REGION Network 16: Odczyt 30011
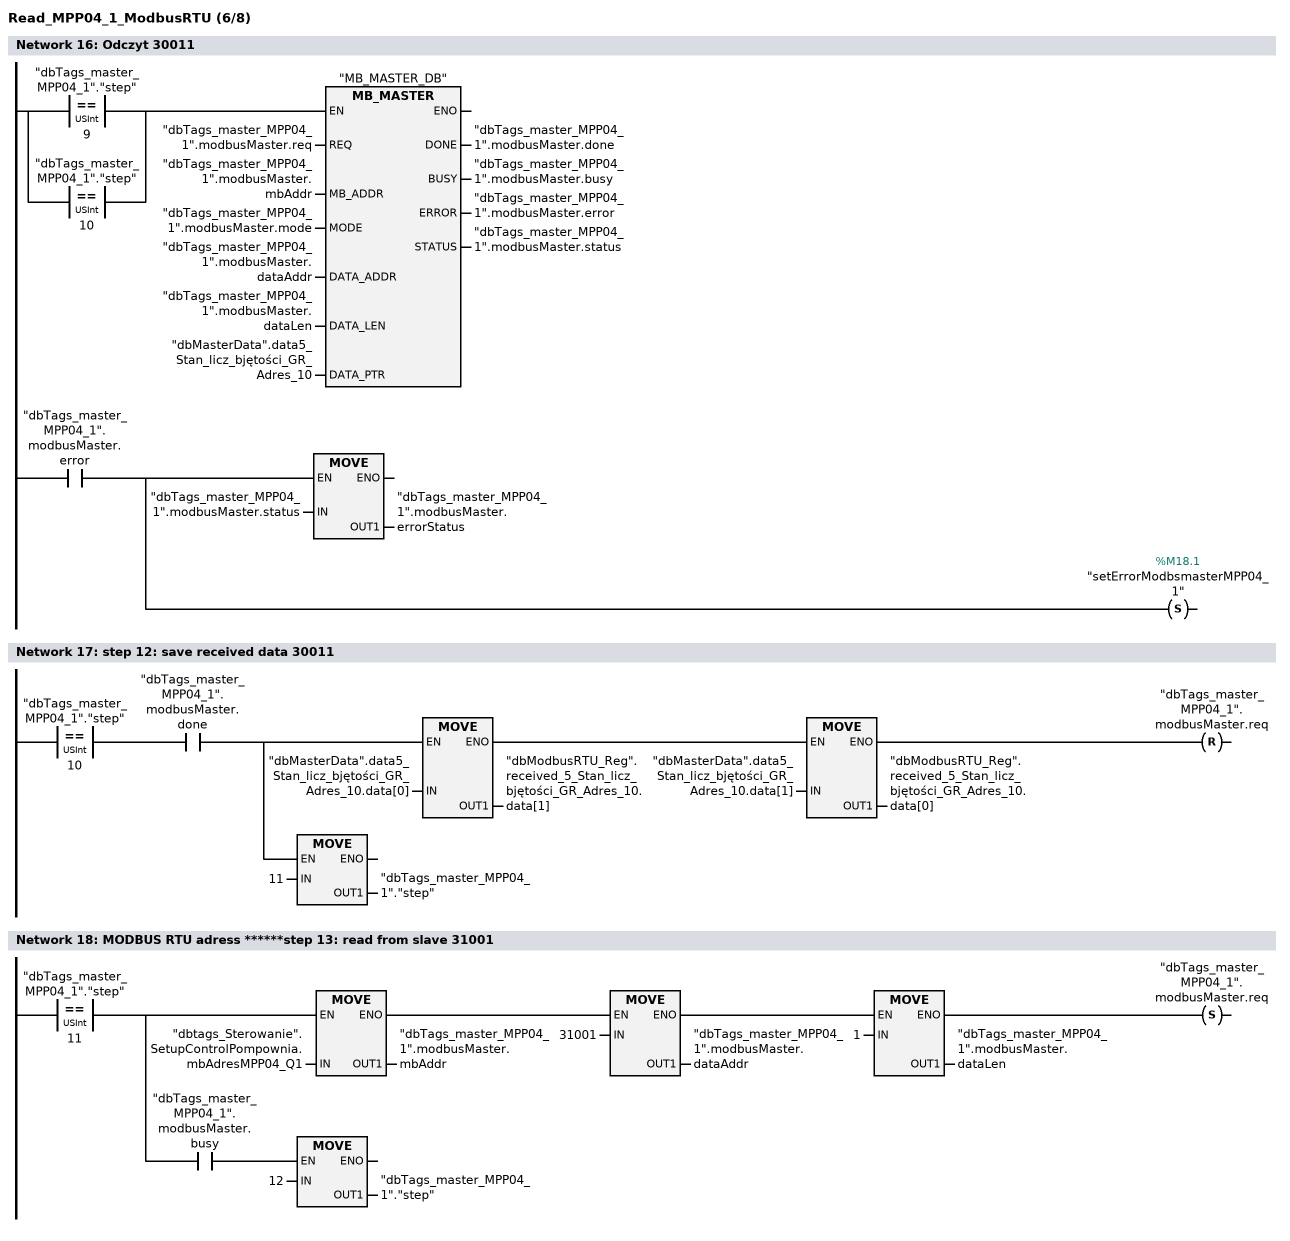
   RUNG wire#powerrail
      { S7_Templates := "SrcType := USInt" } EQ_Contact(in1 := "dbTags_master_MPP04_1"."step", in2 := 9)
      wire#w1
      "MB_MASTER_DB".MB_MASTER(REQ := "dbTags_master_MPP04_1".modbusMaster.req, MB_ADDR := "dbTags_master_MPP04_1".modbusMaster.mbAddr, MODE := "dbTags_master_MPP04_1".modbusMaster.mode, DATA_ADDR := "dbTags_master_MPP04_1".modbusMaster.dataAddr, DATA_LEN := "dbTags_master_MPP04_1".modbusMaster.dataLen, DATA_PTR := "dbMasterData".data5_Stan_licz_bjętości_GR_Adres_10, DONE => "dbTags_master_MPP04_1".modbusMaster.done, BUSY => "dbTags_master_MPP04_1".modbusMaster.busy, ERROR => "dbTags_master_MPP04_1".modbusMaster.error, STATUS => "dbTags_master_MPP04_1".modbusMaster.status)
   END_RUNG
   RUNG wire#powerrail
      { S7_Templates := "SrcType := USInt" } EQ_Contact(in1 := "dbTags_master_MPP04_1"."step", in2 := 10)
   END_RUNG wire#w1
   RUNG wire#powerrail
      Contact( "dbTags_master_MPP04_1".modbusMaster.error )
      wire#w2
      { S7_GenerateENO := "TRUE" } Move(in := "dbTags_master_MPP04_1".modbusMaster.status, out1 => "dbTags_master_MPP04_1".modbusMaster.errorStatus)
   END_RUNG
   RUNG wire#w2
      S_Coil( "setErrorModbsmasterMPP04_1" )
   END_RUNG
   // the same network as SCL:
   IF ("dbTags_master_MPP04_1"."step" = 9) OR ("dbTags_master_MPP04_1"."step" = 10) THEN
       "MB_MASTER_DB"(REQ := "dbTags_master_MPP04_1".modbusMaster.req,   // MB_MASTER
                      MB_ADDR := "dbTags_master_MPP04_1".modbusMaster.mbAddr,
                      MODE := "dbTags_master_MPP04_1".modbusMaster.mode,
                      DATA_ADDR := "dbTags_master_MPP04_1".modbusMaster.dataAddr,
                      DATA_LEN := "dbTags_master_MPP04_1".modbusMaster.dataLen,
                      DATA_PTR := "dbMasterData".data5_Stan_licz_bjętości_GR_Adres_10,
                      DONE => "dbTags_master_MPP04_1".modbusMaster.done,
                      BUSY => "dbTags_master_MPP04_1".modbusMaster.busy,
                      ERROR => "dbTags_master_MPP04_1".modbusMaster.error,
                      STATUS => "dbTags_master_MPP04_1".modbusMaster.status);
   END_IF;
   IF "dbTags_master_MPP04_1".modbusMaster.error THEN
       "dbTags_master_MPP04_1".modbusMaster.errorStatus := "dbTags_master_MPP04_1".modbusMaster.status;
       "setErrorModbsmasterMPP04_1" := TRUE;
   END_IF;
END_REGION

REGION Network 17: step 12: save received data 30011
   RUNG wire#powerrail
      { S7_Templates := "SrcType := USInt" } EQ_Contact(in1 := "dbTags_master_MPP04_1"."step", in2 := 10)
      Contact( "dbTags_master_MPP04_1".modbusMaster.done )
      wire#w1
      { S7_GenerateENO := "TRUE" } Move(in := "dbMasterData".data5_Stan_licz_bjętości_GR_Adres_10.data[0], out1 => "dbModbusRTU_Reg".received_5_Stan_licz_bjętości_GR_Adres_10.data[1])
      { S7_GenerateENO := "TRUE" } Move(in := "dbMasterData".data5_Stan_licz_bjętości_GR_Adres_10.data[1], out1 => "dbModbusRTU_Reg".received_5_Stan_licz_bjętości_GR_Adres_10.data[0])
      R_Coil( "dbTags_master_MPP04_1".modbusMaster.req )
   END_RUNG
   RUNG wire#w1
      { S7_GenerateENO := "TRUE" } Move(in := 11, out1 => "dbTags_master_MPP04_1"."step")
   END_RUNG
   // the same network as SCL:
   // ENO of a box is taken as its EN; it also drops when the box reports an error
   IF ("dbTags_master_MPP04_1"."step" = 10) AND "dbTags_master_MPP04_1".modbusMaster.done THEN
       "dbModbusRTU_Reg".received_5_Stan_licz_bjętości_GR_Adres_10.data[1] := "dbMasterData".data5_Stan_licz_bjętości_GR_Adres_10.data[0];
       "dbModbusRTU_Reg".received_5_Stan_licz_bjętości_GR_Adres_10.data[0] := "dbMasterData".data5_Stan_licz_bjętości_GR_Adres_10.data[1];
       "dbTags_master_MPP04_1".modbusMaster.req := FALSE;
       "dbTags_master_MPP04_1"."step" := 11;
   END_IF;
END_REGION

REGION Network 18: MODBUS RTU adress ******step 13: read from slave 31001
   RUNG wire#powerrail
      { S7_Templates := "SrcType := USInt" } EQ_Contact(in1 := "dbTags_master_MPP04_1"."step", in2 := 11)
      wire#w1
      Move(in := "dbtags_Sterowanie".SetupControlPompownia.mbAdresMPP04_Q1, out1 => "dbTags_master_MPP04_1".modbusMaster.mbAddr)
      { S7_GenerateENO := "TRUE" } Move(in := 31001, out1 => "dbTags_master_MPP04_1".modbusMaster.dataAddr)
      Move(in := 1, out1 => "dbTags_master_MPP04_1".modbusMaster.dataLen)
      S_Coil( "dbTags_master_MPP04_1".modbusMaster.req )
   END_RUNG
   RUNG wire#w1
      Contact( "dbTags_master_MPP04_1".modbusMaster.busy )
      { S7_GenerateENO := "TRUE" } Move(in := 12, out1 => "dbTags_master_MPP04_1"."step")
   END_RUNG
   // the same network as SCL:
   // ENO of a box is taken as its EN; it also drops when the box reports an error
   #_w1 := "dbTags_master_MPP04_1"."step" = 11;
   IF #_w1 THEN
       "dbTags_master_MPP04_1".modbusMaster.mbAddr := "dbtags_Sterowanie".SetupControlPompownia.mbAdresMPP04_Q1;
       "dbTags_master_MPP04_1".modbusMaster.dataAddr := 31001;
       "dbTags_master_MPP04_1".modbusMaster.dataLen := 1;
       "dbTags_master_MPP04_1".modbusMaster.req := TRUE;
   END_IF;
   IF #_w1 AND "dbTags_master_MPP04_1".modbusMaster.busy THEN "dbTags_master_MPP04_1"."step" := 12; END_IF;
END_REGION

REGION Network 19: Odcztyt 31001
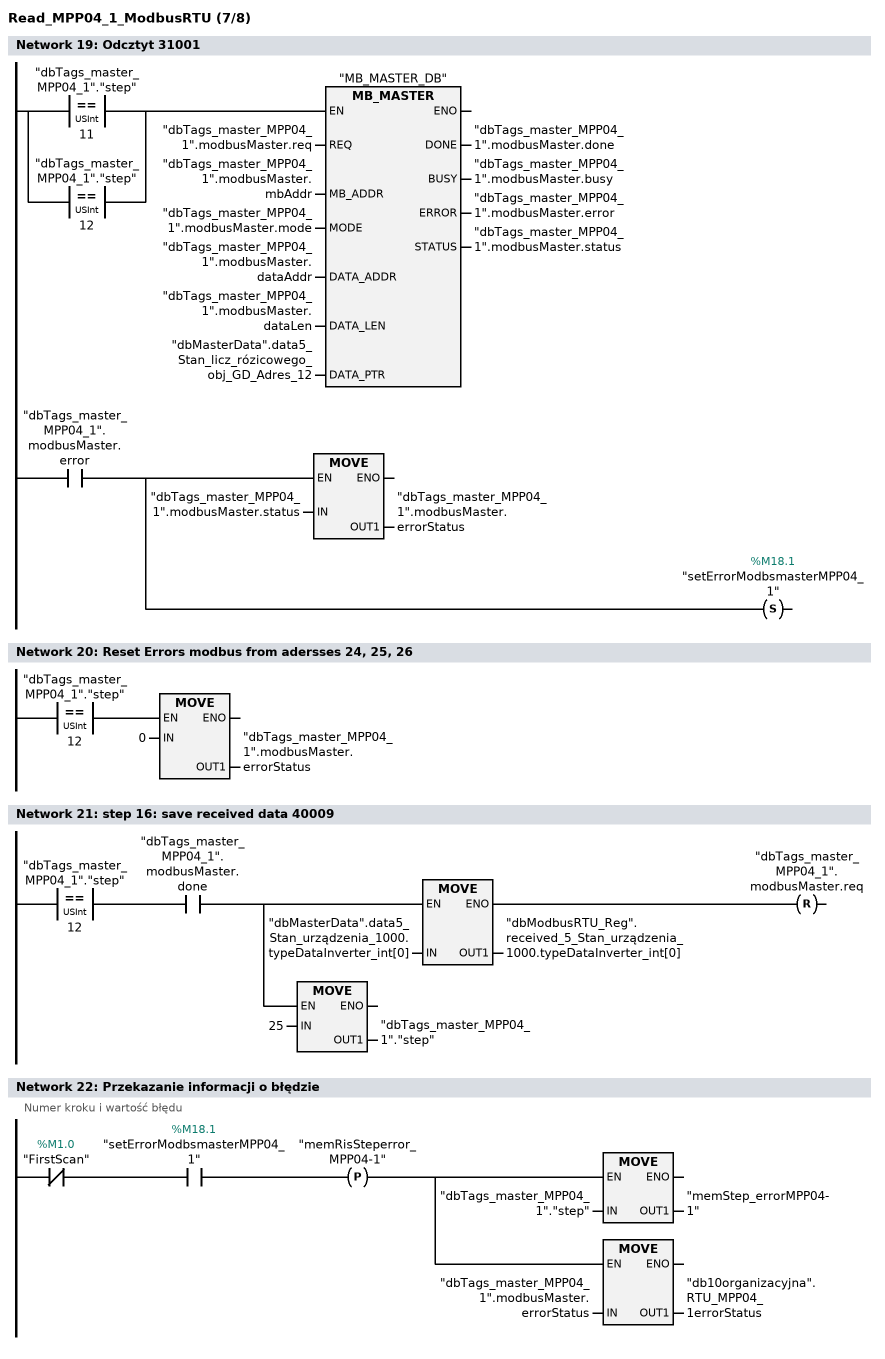
   RUNG wire#powerrail
      { S7_Templates := "SrcType := USInt" } EQ_Contact(in1 := "dbTags_master_MPP04_1"."step", in2 := 11)
      wire#w1
      "MB_MASTER_DB".MB_MASTER(REQ := "dbTags_master_MPP04_1".modbusMaster.req, MB_ADDR := "dbTags_master_MPP04_1".modbusMaster.mbAddr, MODE := "dbTags_master_MPP04_1".modbusMaster.mode, DATA_ADDR := "dbTags_master_MPP04_1".modbusMaster.dataAddr, DATA_LEN := "dbTags_master_MPP04_1".modbusMaster.dataLen, DATA_PTR := "dbMasterData".data5_Stan_licz_rózicowego_obj_GD_Adres_12, DONE => "dbTags_master_MPP04_1".modbusMaster.done, BUSY => "dbTags_master_MPP04_1".modbusMaster.busy, ERROR => "dbTags_master_MPP04_1".modbusMaster.error, STATUS => "dbTags_master_MPP04_1".modbusMaster.status)
   END_RUNG
   RUNG wire#powerrail
      { S7_Templates := "SrcType := USInt" } EQ_Contact(in1 := "dbTags_master_MPP04_1"."step", in2 := 12)
   END_RUNG wire#w1
   RUNG wire#powerrail
      Contact( "dbTags_master_MPP04_1".modbusMaster.error )
      wire#w2
      { S7_GenerateENO := "TRUE" } Move(in := "dbTags_master_MPP04_1".modbusMaster.status, out1 => "dbTags_master_MPP04_1".modbusMaster.errorStatus)
   END_RUNG
   RUNG wire#w2
      S_Coil( "setErrorModbsmasterMPP04_1" )
   END_RUNG
   // the same network as SCL:
   IF ("dbTags_master_MPP04_1"."step" = 11) OR ("dbTags_master_MPP04_1"."step" = 12) THEN
       "MB_MASTER_DB"(REQ := "dbTags_master_MPP04_1".modbusMaster.req,   // MB_MASTER
                      MB_ADDR := "dbTags_master_MPP04_1".modbusMaster.mbAddr,
                      MODE := "dbTags_master_MPP04_1".modbusMaster.mode,
                      DATA_ADDR := "dbTags_master_MPP04_1".modbusMaster.dataAddr,
                      DATA_LEN := "dbTags_master_MPP04_1".modbusMaster.dataLen,
                      DATA_PTR := "dbMasterData".data5_Stan_licz_rózicowego_obj_GD_Adres_12,
                      DONE => "dbTags_master_MPP04_1".modbusMaster.done,
                      BUSY => "dbTags_master_MPP04_1".modbusMaster.busy,
                      ERROR => "dbTags_master_MPP04_1".modbusMaster.error,
                      STATUS => "dbTags_master_MPP04_1".modbusMaster.status);
   END_IF;
   IF "dbTags_master_MPP04_1".modbusMaster.error THEN
       "dbTags_master_MPP04_1".modbusMaster.errorStatus := "dbTags_master_MPP04_1".modbusMaster.status;
       "setErrorModbsmasterMPP04_1" := TRUE;
   END_IF;
END_REGION

REGION Network 20: Reset Errors modbus from adersses 24, 25, 26
   RUNG wire#powerrail
      { S7_Templates := "SrcType := USInt" } EQ_Contact(in1 := "dbTags_master_MPP04_1"."step", in2 := 12)
      { S7_GenerateENO := "TRUE" } Move(in := 0, out1 => "dbTags_master_MPP04_1".modbusMaster.errorStatus)
   END_RUNG
   // the same network as SCL:
   IF "dbTags_master_MPP04_1"."step" = 12 THEN "dbTags_master_MPP04_1".modbusMaster.errorStatus := 0; END_IF;
END_REGION

REGION Network 21: step 16: save received data 40009
   RUNG wire#powerrail
      { S7_Templates := "SrcType := USInt" } EQ_Contact(in1 := "dbTags_master_MPP04_1"."step", in2 := 12)
      Contact( "dbTags_master_MPP04_1".modbusMaster.done )
      wire#w1
      { S7_GenerateENO := "TRUE" } Move(in := "dbMasterData".data5_Stan_urządzenia_1000.typeDataInverter_int[0], out1 => "dbModbusRTU_Reg".received_5_Stan_urządzenia_1000.typeDataInverter_int[0])
      R_Coil( "dbTags_master_MPP04_1".modbusMaster.req )
   END_RUNG
   RUNG wire#w1
      { S7_GenerateENO := "TRUE" } Move(in := 25, out1 => "dbTags_master_MPP04_1"."step")
   END_RUNG
   // the same network as SCL:
   // ENO of a box is taken as its EN; it also drops when the box reports an error
   IF ("dbTags_master_MPP04_1"."step" = 12) AND "dbTags_master_MPP04_1".modbusMaster.done THEN
       "dbModbusRTU_Reg".received_5_Stan_urządzenia_1000.typeDataInverter_int[0] := "dbMasterData".data5_Stan_urządzenia_1000.typeDataInverter_int[0];
       "dbTags_master_MPP04_1".modbusMaster.req := FALSE;
       "dbTags_master_MPP04_1"."step" := 25;
   END_IF;
END_REGION

REGION Network 22: Przekazanie informacji o błędzie
   // Numer kroku i wartość błędu
   RUNG wire#powerrail
      I_Contact( "FirstScan" )
      Contact( "setErrorModbsmasterMPP04_1" )
      P_Trig( "memRisSteperror_MPP04-1" )
      wire#w1
      Move(in := "dbTags_master_MPP04_1"."step", out1 => "memStep_errorMPP04-1")
   END_RUNG
   RUNG wire#w1
      { S7_GenerateENO := "TRUE" } Move(in := "dbTags_master_MPP04_1".modbusMaster.errorStatus, out1 => "db10organizacyjna".RTU_MPP04_1errorStatus)
   END_RUNG
   // the same network as SCL:
   #_w1 := NOT "FirstScan" AND "setErrorModbsmasterMPP04_1";
   #_w2 := #_w1 AND NOT "memRisSteperror_MPP04-1";   // rising edge
   "memRisSteperror_MPP04-1" := #_w1;
   IF #_w2 THEN
       "memStep_errorMPP04-1" := "dbTags_master_MPP04_1"."step";
       "db10organizacyjna".RTU_MPP04_1errorStatus := "dbTags_master_MPP04_1".modbusMaster.errorStatus;
   END_IF;
END_REGION

REGION Network 23: Obsługa błędów Modbaus
   // Inicjacja pętli modbus dla następnego urządzenia
   // Ustawienie kroku pętli na stan awaria [27]
   // Uwolnienie linni modbus
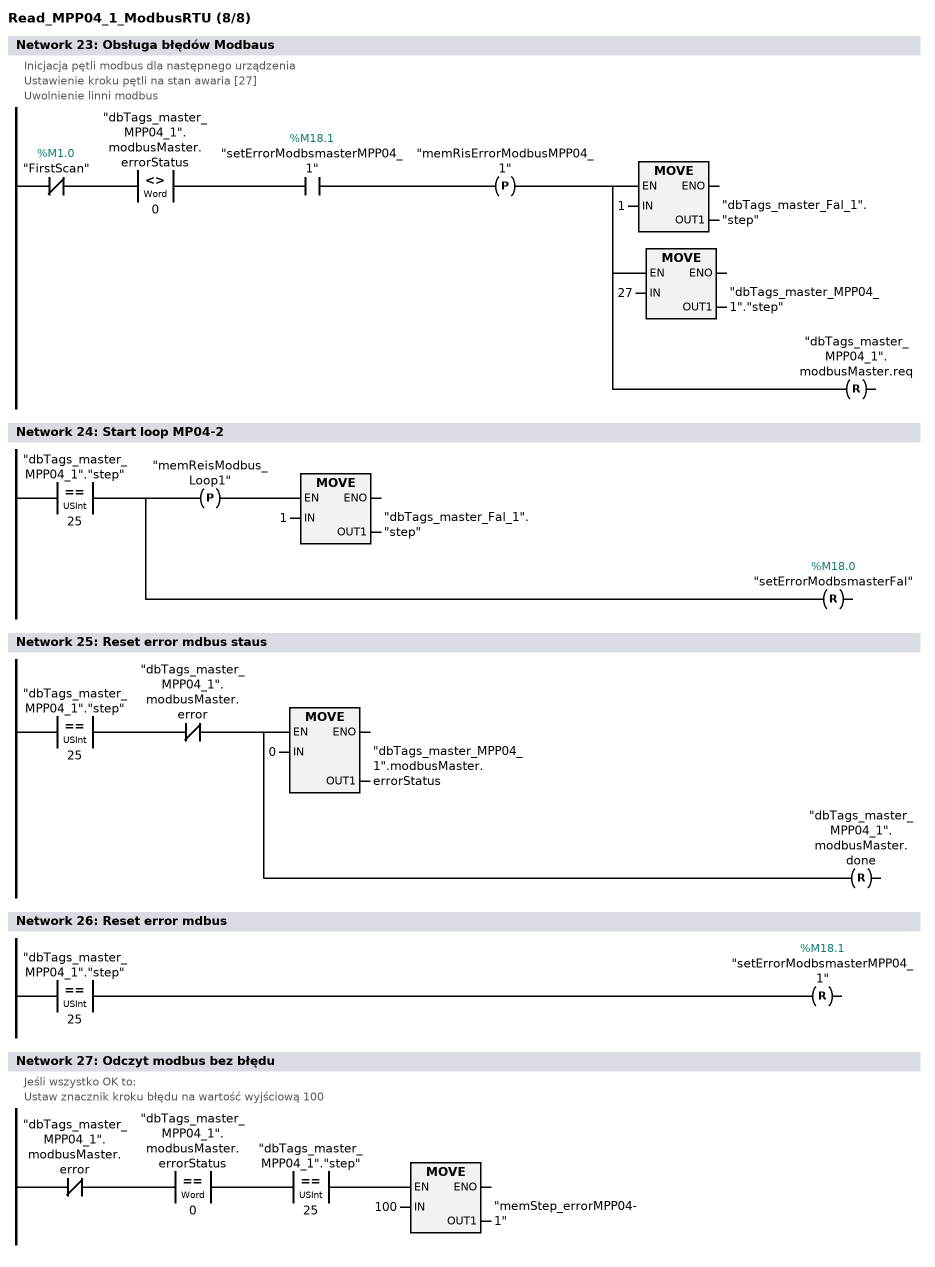
   RUNG wire#powerrail
      I_Contact( "FirstScan" )
      { S7_Templates := "SrcType := Word" } NE_Contact(in1 := "dbTags_master_MPP04_1".modbusMaster.errorStatus, in2 := 0)
      Contact( "setErrorModbsmasterMPP04_1" )
      P_Trig( "memRisErrorModbusMPP04_1" )
      wire#w1
      { S7_GenerateENO := "TRUE" } Move(in := 1, out1 => "dbTags_master_Fal_1"."step")
   END_RUNG
   RUNG wire#w1
      { S7_GenerateENO := "TRUE" } Move(in := 27, out1 => "dbTags_master_MPP04_1"."step")
   END_RUNG
   RUNG wire#w1
      R_Coil( "dbTags_master_MPP04_1".modbusMaster.req )
   END_RUNG
   // the same network as SCL:
   #_w1 := NOT "FirstScan" AND ("dbTags_master_MPP04_1".modbusMaster.errorStatus <> 0) AND "setErrorModbsmasterMPP04_1";
   #_w2 := #_w1 AND NOT "memRisErrorModbusMPP04_1";   // rising edge
   "memRisErrorModbusMPP04_1" := #_w1;
   IF #_w2 THEN
       "dbTags_master_Fal_1"."step" := 1;
       "dbTags_master_MPP04_1"."step" := 27;
       "dbTags_master_MPP04_1".modbusMaster.req := FALSE;
   END_IF;
END_REGION

REGION Network 24: Start loop MP04-2
   RUNG wire#powerrail
      { S7_Templates := "SrcType := USInt" } EQ_Contact(in1 := "dbTags_master_MPP04_1"."step", in2 := 25)
      wire#w1
      P_Trig( "memReisModbus_Loop1" )
      { S7_GenerateENO := "TRUE" } Move(in := 1, out1 => "dbTags_master_Fal_1"."step")
   END_RUNG
   RUNG wire#w1
      R_Coil( "setErrorModbsmasterFal" )
   END_RUNG
   // the same network as SCL:
   #_w1 := "dbTags_master_MPP04_1"."step" = 25;
   #_w2 := #_w1 AND NOT "memReisModbus_Loop1";   // rising edge
   "memReisModbus_Loop1" := #_w1;
   IF #_w2 THEN "dbTags_master_Fal_1"."step" := 1; END_IF;
   IF #_w1 THEN "setErrorModbsmasterFal" := FALSE; END_IF;
END_REGION

REGION Network 25: Reset error mdbus staus
   RUNG wire#powerrail
      { S7_Templates := "SrcType := USInt" } EQ_Contact(in1 := "dbTags_master_MPP04_1"."step", in2 := 25)
      I_Contact( "dbTags_master_MPP04_1".modbusMaster.error )
      wire#w1
      { S7_GenerateENO := "TRUE" } Move(in := 0, out1 => "dbTags_master_MPP04_1".modbusMaster.errorStatus)
   END_RUNG
   RUNG wire#w1
      R_Coil( "dbTags_master_MPP04_1".modbusMaster.done )
   END_RUNG
   // the same network as SCL:
   IF ("dbTags_master_MPP04_1"."step" = 25) AND NOT "dbTags_master_MPP04_1".modbusMaster.error THEN
       "dbTags_master_MPP04_1".modbusMaster.errorStatus := 0;
       "dbTags_master_MPP04_1".modbusMaster.done := FALSE;
   END_IF;
END_REGION

REGION Network 26: Reset error mdbus
   RUNG wire#powerrail
      { S7_Templates := "SrcType := USInt" } EQ_Contact(in1 := "dbTags_master_MPP04_1"."step", in2 := 25)
      R_Coil( "setErrorModbsmasterMPP04_1" )
   END_RUNG
   // the same network as SCL:
   IF "dbTags_master_MPP04_1"."step" = 25 THEN "setErrorModbsmasterMPP04_1" := FALSE; END_IF;
END_REGION

REGION Network 27: Odczyt modbus bez błędu
   // Jeśli wszystko OK to:
   // Ustaw znacznik kroku błędu na wartość wyjściową 100
   RUNG wire#powerrail
      I_Contact( "dbTags_master_MPP04_1".modbusMaster.error )
      { S7_Templates := "SrcType := Word" } EQ_Contact(in1 := "dbTags_master_MPP04_1".modbusMaster.errorStatus, in2 := 0)
      { S7_Templates := "SrcType := USInt" } EQ_Contact(in1 := "dbTags_master_MPP04_1"."step", in2 := 25)
      { S7_GenerateENO := "TRUE" } Move(in := 100, out1 => "memStep_errorMPP04-1")
   END_RUNG
   // the same network as SCL:
   IF NOT "dbTags_master_MPP04_1".modbusMaster.error AND ("dbTags_master_MPP04_1".modbusMaster.errorStatus = 0) AND ("dbTags_master_MPP04_1"."step" = 25) THEN
       "memStep_errorMPP04-1" := 100;
   END_IF;
END_REGION
END_FUNCTION

FUNCTION_BLOCK "Write_dbHold_TCP_Sending"
{ S7_Optimized_Access := 'TRUE' }
VERSION : 0.1

BEGIN
	(*
	
	*)
	
	
	
	
	REGION Strategia Sterowania Pompownią 
	  // przekazanie wartości do PLC2 Zbiorniki
	  "dbHold_RRG".Sending.set_strategia_sterowania:= "dbHoldRegSlave_to_MT101".instSygSter_1;
	  
	END_REGION
	
	REGION _name_
	  // 
	
	
	  
	  
	END_REGION
	
	
	
END_FUNCTION_BLOCK

FUNCTION "Blok liczników pracy" : Void   // FC8, LAD
TITLE = Wywołanie funkcji liczników pracy
{ S7_Optimized_Access := 'TRUE' }
AUTHOR : RTecmer
VERSION : 0.1
// Funkcja wywołuje liczniki pracy napędów
// stored: AutoNumber true, IsIECCheckEnabled false, SetENOAutomatically false, UDAEnableTagReadback false
BEGIN

REGION Network 1: Pompa P1
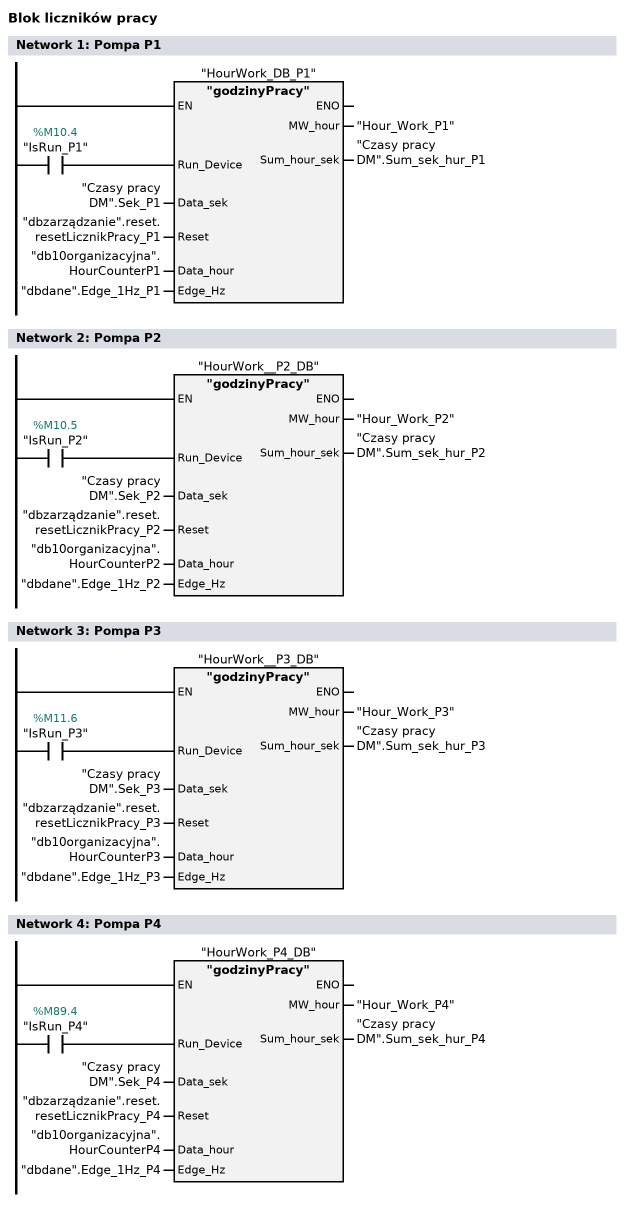
   RUNG wire#powerrail
      "HourWork_DB_P1"(Run_Device := wire#w1, Data_sek := "Czasy pracy DM".Sek_P1, Reset := "dbzarządzanie".reset.resetLicznikPracy_P1, Data_hour := "db10organizacyjna".HourCounterP1, Edge_Hz := "dbdane".Edge_1Hz_P1, MW_hour => "Hour_Work_P1", Sum_hour_sek => "Czasy pracy DM".Sum_sek_hur_P1)
   END_RUNG
   RUNG wire#powerrail
      Contact( "IsRun_P1" )
   END_RUNG wire#w1
   // the same network as SCL:
   "HourWork_DB_P1"(Run_Device := "IsRun_P1",   // "godzinyPracy"
                    Data_sek := "Czasy pracy DM".Sek_P1,
                    Reset := "dbzarządzanie".reset.resetLicznikPracy_P1,
                    Data_hour := "db10organizacyjna".HourCounterP1,
                    Edge_Hz := "dbdane".Edge_1Hz_P1,
                    MW_hour => "Hour_Work_P1",
                    Sum_hour_sek => "Czasy pracy DM".Sum_sek_hur_P1);
END_REGION

REGION Network 2: Pompa P2
   RUNG wire#powerrail
      "HourWork__P2_DB"(Run_Device := wire#w1, Data_sek := "Czasy pracy DM".Sek_P2, Reset := "dbzarządzanie".reset.resetLicznikPracy_P2, Data_hour := "db10organizacyjna".HourCounterP2, Edge_Hz := "dbdane".Edge_1Hz_P2, MW_hour => "Hour_Work_P2", Sum_hour_sek => "Czasy pracy DM".Sum_sek_hur_P2)
   END_RUNG
   RUNG wire#powerrail
      Contact( "IsRun_P2" )
   END_RUNG wire#w1
   // the same network as SCL:
   "HourWork__P2_DB"(Run_Device := "IsRun_P2",   // "godzinyPracy"
                     Data_sek := "Czasy pracy DM".Sek_P2,
                     Reset := "dbzarządzanie".reset.resetLicznikPracy_P2,
                     Data_hour := "db10organizacyjna".HourCounterP2,
                     Edge_Hz := "dbdane".Edge_1Hz_P2,
                     MW_hour => "Hour_Work_P2",
                     Sum_hour_sek => "Czasy pracy DM".Sum_sek_hur_P2);
END_REGION

REGION Network 3: Pompa P3
   RUNG wire#powerrail
      "HourWork__P3_DB"(Run_Device := wire#w1, Data_sek := "Czasy pracy DM".Sek_P3, Reset := "dbzarządzanie".reset.resetLicznikPracy_P3, Data_hour := "db10organizacyjna".HourCounterP3, Edge_Hz := "dbdane".Edge_1Hz_P3, MW_hour => "Hour_Work_P3", Sum_hour_sek => "Czasy pracy DM".Sum_sek_hur_P3)
   END_RUNG
   RUNG wire#powerrail
      Contact( "IsRun_P3" )
   END_RUNG wire#w1
   // the same network as SCL:
   "HourWork__P3_DB"(Run_Device := "IsRun_P3",   // "godzinyPracy"
                     Data_sek := "Czasy pracy DM".Sek_P3,
                     Reset := "dbzarządzanie".reset.resetLicznikPracy_P3,
                     Data_hour := "db10organizacyjna".HourCounterP3,
                     Edge_Hz := "dbdane".Edge_1Hz_P3,
                     MW_hour => "Hour_Work_P3",
                     Sum_hour_sek => "Czasy pracy DM".Sum_sek_hur_P3);
END_REGION

REGION Network 4: Pompa P4
   RUNG wire#powerrail
      "HourWork_P4_DB"(Run_Device := wire#w1, Data_sek := "Czasy pracy DM".Sek_P4, Reset := "dbzarządzanie".reset.resetLicznikPracy_P4, Data_hour := "db10organizacyjna".HourCounterP4, Edge_Hz := "dbdane".Edge_1Hz_P4, MW_hour => "Hour_Work_P4", Sum_hour_sek => "Czasy pracy DM".Sum_sek_hur_P4)
   END_RUNG
   RUNG wire#powerrail
      Contact( "IsRun_P4" )
   END_RUNG wire#w1
   // the same network as SCL:
   "HourWork_P4_DB"(Run_Device := "IsRun_P4",   // "godzinyPracy"
                    Data_sek := "Czasy pracy DM".Sek_P4,
                    Reset := "dbzarządzanie".reset.resetLicznikPracy_P4,
                    Data_hour := "db10organizacyjna".HourCounterP4,
                    Edge_Hz := "dbdane".Edge_1Hz_P4,
                    MW_hour => "Hour_Work_P4",
                    Sum_hour_sek => "Czasy pracy DM".Sum_sek_hur_P4);
END_REGION
END_FUNCTION

FUNCTION_BLOCK "godzinyPracy"   // FB2, LAD
{ S7_Optimized_Access := 'TRUE' }
AUTHOR : RTecmer
FAMILY : XMHour
VERSION : 0.1
// Licznik czasu pracy
// stored: AutoNumber true, IsIECCheckEnabled false, IsRetainMemResEnabled false, MemoryReserve 500, SetENOAutomatically false, UDAEnableTagReadback false
   VAR_INPUT
      Run_Device : Bool;
   END_VAR
   VAR_OUTPUT
      MW_hour : DWord;
      Sum_hour_sek : Real;   // Licznik sumator godzin i sekund na potrzeby wyznaczania dumchawy do pracy
   END_VAR
   VAR_IN_OUT
      Data_sek : Int;
      Reset { ExternalAccessible := 'False'; ExternalVisible := 'False'; ExternalWritable := 'False'} : Bool;
      Data_hour : DWord;
      Edge_Hz { ExternalAccessible := 'False'; ExternalVisible := 'False'; ExternalWritable := 'False'} : Bool;
   END_VAR
   VAR
      sek_real { ExternalAccessible := 'False'; ExternalVisible := 'False'; ExternalWritable := 'False'} : Real;   // pomocnicza konwerski sekund
      actSekReal { ExternalAccessible := 'False'; ExternalVisible := 'False'; ExternalWritable := 'False'} : Real;   // aktualne sekundy po konwersji
      hour_sek { ExternalAccessible := 'False'; ExternalVisible := 'False'; ExternalWritable := 'False'} : Real;
   END_VAR
   VAR_TEMP   // added for the SCL form of the ladder/FBD networks
      _w1 : Bool;
      _w2 : Bool;
   END_VAR
BEGIN

REGION Network 1
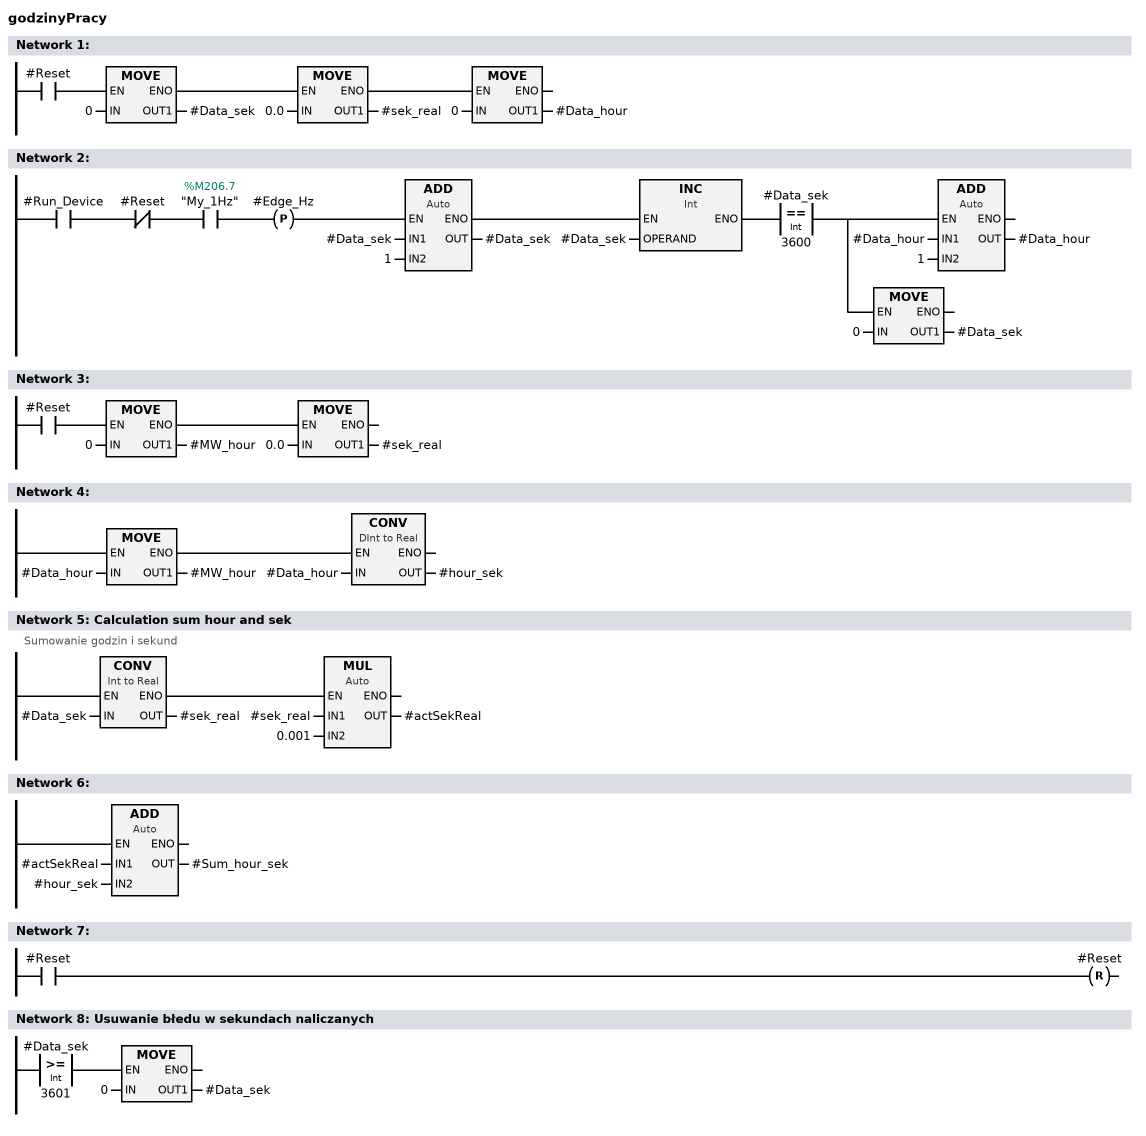
   RUNG wire#powerrail
      Contact( #Reset )
      { S7_GenerateENO := "TRUE" } Move(in := 0, out1 => #Data_sek)
      { S7_GenerateENO := "TRUE" } Move(in := 0.0, out1 => #sek_real)
      { S7_GenerateENO := "TRUE" } Move(in := 0, out1 => #Data_hour)
   END_RUNG
   // the same network as SCL:
   // ENO of a box is taken as its EN; it also drops when the box reports an error
   IF #Reset THEN
       #Data_sek := 0;
       #sek_real := 0.0;
       #Data_hour := 0;
   END_IF;
END_REGION

REGION Network 2
   RUNG wire#powerrail
      Contact( #Run_Device )
      I_Contact( #Reset )
      Contact( "My_1Hz" )
      P_Trig( #Edge_Hz )
      { S7_GenerateENO := "TRUE" } Add(in1 := #Data_sek, in2 := 1, out => #Data_sek)
      { S7_Templates := "DestType := Int"; S7_GenerateENO := "TRUE" } Inc( #Data_sek )
      { S7_Templates := "SrcType := Int" } EQ_Contact(in1 := #Data_sek, in2 := 3600)
      wire#w1
      { S7_GenerateENO := "TRUE" } Add(in1 := #Data_hour, in2 := 1, out => #Data_hour)
   END_RUNG
   RUNG wire#w1
      { S7_GenerateENO := "TRUE" } Move(in := 0, out1 => #Data_sek)
   END_RUNG
   // the same network as SCL:
   // ENO of a box is taken as its EN; it also drops when the box reports an error
   #_w1 := #Run_Device AND NOT #Reset AND "My_1Hz";
   #_w2 := #_w1 AND NOT #Edge_Hz;   // rising edge
   #Edge_Hz := #_w1;
   IF #_w2 THEN
       #Data_sek := #Data_sek + 1;
       #Data_sek := #Data_sek + 1;
   END_IF;
   IF #_w2 AND (#Data_sek = 3600) THEN
       #Data_hour := #Data_hour + 1;
       #Data_sek := 0;
   END_IF;
END_REGION

REGION Network 3
   RUNG wire#powerrail
      Contact( #Reset )
      { S7_GenerateENO := "TRUE" } Move(in := 0, out1 => #MW_hour)
      { S7_GenerateENO := "TRUE" } Move(in := 0.0, out1 => #sek_real)
   END_RUNG
   // the same network as SCL:
   // ENO of a box is taken as its EN; it also drops when the box reports an error
   IF #Reset THEN
       #MW_hour := 0;
       #sek_real := 0.0;
   END_IF;
END_REGION

REGION Network 4
   RUNG wire#powerrail
      { S7_GenerateENO := "TRUE" } Move(in := #Data_hour, out1 => #MW_hour)
      { S7_Templates := "[SrcType := DInt, DestType := Real]" } Convert(in := #Data_hour, out => #hour_sek)
   END_RUNG
   // the same network as SCL:
   // ENO of a box is taken as its EN; it also drops when the box reports an error
   #MW_hour := #Data_hour;
   #hour_sek := DINT_TO_REAL(#Data_hour);
END_REGION

REGION Network 5: Calculation sum hour and sek
   // Sumowanie godzin i sekund
   RUNG wire#powerrail
      { S7_Templates := "[SrcType := Int, DestType := Real]" } Convert(in := #Data_sek, out => #sek_real)
      Mul(in1 := #sek_real, in2 := 0.001, out => #actSekReal)
   END_RUNG
   // the same network as SCL:
   #sek_real := INT_TO_REAL(#Data_sek);
   #actSekReal := #sek_real * 0.001;
END_REGION

REGION Network 6
   RUNG wire#powerrail
      Add(in1 := #actSekReal, in2 := #hour_sek, out => #Sum_hour_sek)
   END_RUNG
   // the same network as SCL:
   #Sum_hour_sek := #actSekReal + #hour_sek;
END_REGION

REGION Network 7
   RUNG wire#powerrail
      Contact( #Reset )
      R_Coil( #Reset )
   END_RUNG
   // the same network as SCL:
   IF #Reset THEN #Reset := FALSE; END_IF;
END_REGION

REGION Network 8: Usuwanie błedu w sekundach naliczanych
   RUNG wire#powerrail
      { S7_Templates := "SrcType := Int" } GE_Contact(in1 := #Data_sek, in2 := 3601)
      { S7_GenerateENO := "TRUE" } Move(in := 0, out1 => #Data_sek)
   END_RUNG
   // the same network as SCL:
   IF #Data_sek >= 3601 THEN #Data_sek := 0; END_IF;
END_REGION
END_FUNCTION_BLOCK

FUNCTION "Wybór_pompy_najmniej godzin" : Void   // FC17, LAD
TITLE = Selektor godzin pracy / Compressor selection from hours
{ S7_Optimized_Access := 'TRUE' }
AUTHOR : rtecmer
VERSION : 0.1
// Ustawienie kolejności wyboru pomp z wyrównaniem czasu pracy. Podstawa najmniejsza ilość godzin pracy / Ustawienie kolejności wyboru kompresorów z wyrównaniem czasu pracy. Podstawa najmniejsza ilość godzin pracy
// stored: AutoNumber true, IsIECCheckEnabled false, SetENOAutomatically false, UDAEnableTagReadback false
   VAR_IN_OUT
      Reset : Bool;   // Reset po błędzie
   END_VAR
   VAR_TEMP
      tmp_Sum_sek_P1 : Int;   // tymczasowy licznik sumy sekund
      tmp_Sum_sek_P2 : Int;   // tymczasowy licznik sumy sekund
      tmp_Sum_sek_P3 : Int;   // tymczasowy licznik sumy sekund
      tmp_Sum_sek_P4 : Int;   // tymczasowy licznik sumy sekund
   END_VAR
BEGIN

REGION Network 1: Reakcja na równe liczniki
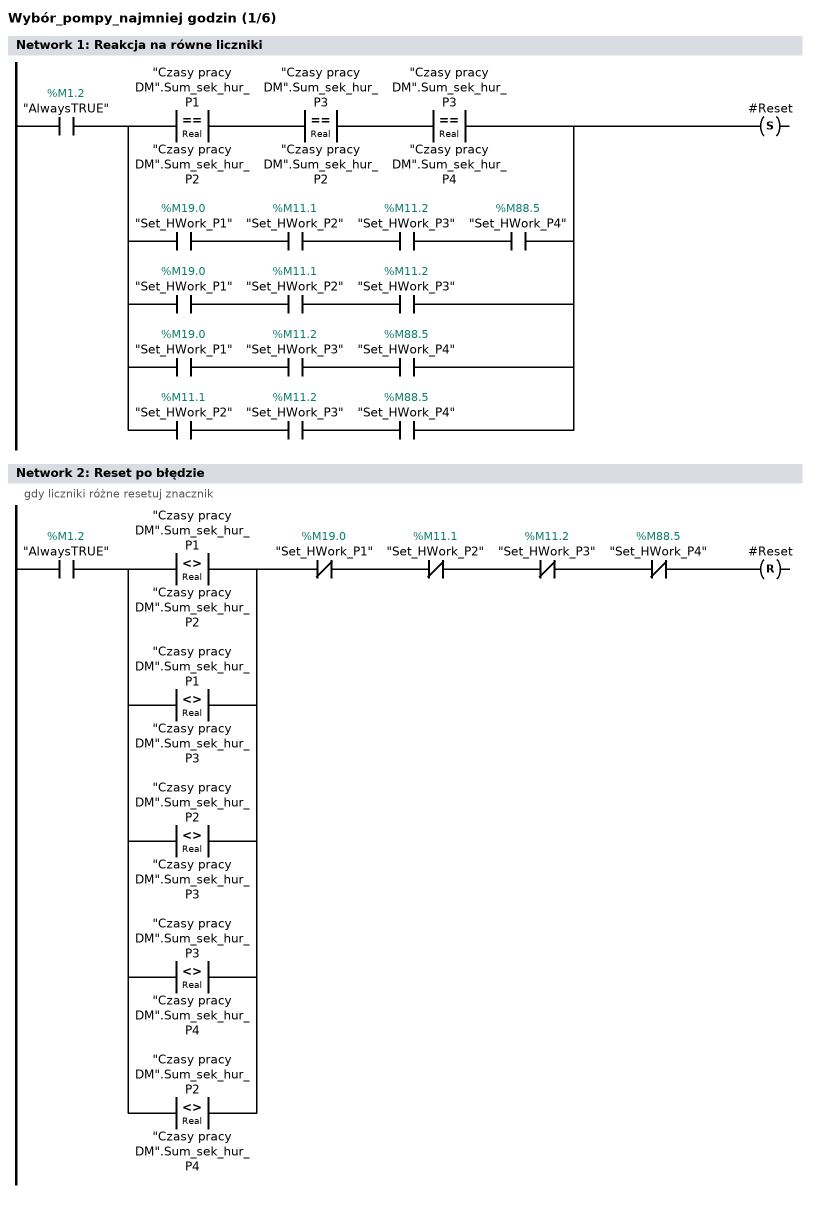
   RUNG wire#powerrail
      Contact( "AlwaysTRUE" )
      wire#w1
      { S7_Templates := "SrcType := Real" } EQ_Contact(in1 := "Czasy pracy DM".Sum_sek_hur_P1, in2 := "Czasy pracy DM".Sum_sek_hur_P2)
      { S7_Templates := "SrcType := Real" } EQ_Contact(in1 := "Czasy pracy DM".Sum_sek_hur_P3, in2 := "Czasy pracy DM".Sum_sek_hur_P2)
      { S7_Templates := "SrcType := Real" } EQ_Contact(in1 := "Czasy pracy DM".Sum_sek_hur_P3, in2 := "Czasy pracy DM".Sum_sek_hur_P4)
      wire#w2
      S_Coil( #Reset )
   END_RUNG
   RUNG wire#w1
      Contact( "Set_HWork_P1" )
      Contact( "Set_HWork_P2" )
      Contact( "Set_HWork_P3" )
      Contact( "Set_HWork_P4" )
   END_RUNG wire#w2
   RUNG wire#w1
      Contact( "Set_HWork_P1" )
      Contact( "Set_HWork_P2" )
      Contact( "Set_HWork_P3" )
   END_RUNG wire#w2
   RUNG wire#w1
      Contact( "Set_HWork_P1" )
      Contact( "Set_HWork_P3" )
      Contact( "Set_HWork_P4" )
   END_RUNG wire#w2
   RUNG wire#w1
      Contact( "Set_HWork_P2" )
      Contact( "Set_HWork_P3" )
      Contact( "Set_HWork_P4" )
   END_RUNG wire#w2
   // the same network as SCL:
   IF "AlwaysTRUE" AND ((("Czasy pracy DM".Sum_sek_hur_P1 = "Czasy pracy DM".Sum_sek_hur_P2) AND ("Czasy pracy DM".Sum_sek_hur_P3 = "Czasy pracy DM".Sum_sek_hur_P2) AND ("Czasy pracy DM".Sum_sek_hur_P3 = "Czasy pracy DM".Sum_sek_hur_P4)) OR ("Set_HWork_P1" AND "Set_HWork_P2" AND "Set_HWork_P3" AND "Set_HWork_P4") OR ("Set_HWork_P1" AND "Set_HWork_P2" AND "Set_HWork_P3") OR ("Set_HWork_P1" AND "Set_HWork_P3" AND "Set_HWork_P4") OR ("Set_HWork_P2" AND "Set_HWork_P3" AND "Set_HWork_P4")) THEN
       #Reset := TRUE;
   END_IF;
END_REGION

REGION Network 2: Reset po błędzie
   // gdy liczniki różne resetuj znacznik
   RUNG wire#powerrail
      Contact( "AlwaysTRUE" )
      wire#w1
      { S7_Templates := "SrcType := Real" } NE_Contact(in1 := "Czasy pracy DM".Sum_sek_hur_P1, in2 := "Czasy pracy DM".Sum_sek_hur_P2)
      wire#w2
      I_Contact( "Set_HWork_P1" )
      I_Contact( "Set_HWork_P2" )
      I_Contact( "Set_HWork_P3" )
      I_Contact( "Set_HWork_P4" )
      R_Coil( #Reset )
   END_RUNG
   RUNG wire#w1
      { S7_Templates := "SrcType := Real" } NE_Contact(in1 := "Czasy pracy DM".Sum_sek_hur_P1, in2 := "Czasy pracy DM".Sum_sek_hur_P3)
   END_RUNG wire#w2
   RUNG wire#w1
      { S7_Templates := "SrcType := Real" } NE_Contact(in1 := "Czasy pracy DM".Sum_sek_hur_P2, in2 := "Czasy pracy DM".Sum_sek_hur_P3)
   END_RUNG wire#w2
   RUNG wire#w1
      { S7_Templates := "SrcType := Real" } NE_Contact(in1 := "Czasy pracy DM".Sum_sek_hur_P3, in2 := "Czasy pracy DM".Sum_sek_hur_P4)
   END_RUNG wire#w2
   RUNG wire#w1
      { S7_Templates := "SrcType := Real" } NE_Contact(in1 := "Czasy pracy DM".Sum_sek_hur_P2, in2 := "Czasy pracy DM".Sum_sek_hur_P4)
   END_RUNG wire#w2
   // the same network as SCL:
   IF "AlwaysTRUE" AND (("Czasy pracy DM".Sum_sek_hur_P1 <> "Czasy pracy DM".Sum_sek_hur_P2) OR ("Czasy pracy DM".Sum_sek_hur_P1 <> "Czasy pracy DM".Sum_sek_hur_P3) OR ("Czasy pracy DM".Sum_sek_hur_P2 <> "Czasy pracy DM".Sum_sek_hur_P3) OR ("Czasy pracy DM".Sum_sek_hur_P3 <> "Czasy pracy DM".Sum_sek_hur_P4) OR ("Czasy pracy DM".Sum_sek_hur_P2 <> "Czasy pracy DM".Sum_sek_hur_P4)) AND NOT "Set_HWork_P1" AND NOT "Set_HWork_P2" AND NOT "Set_HWork_P3" AND NOT "Set_HWork_P4" THEN
       #Reset := FALSE;
   END_IF;
END_REGION

REGION Network 3: Reset znaczników aktywacji napędu od czasu pracy / Wyłączenie napedów od równych liczników
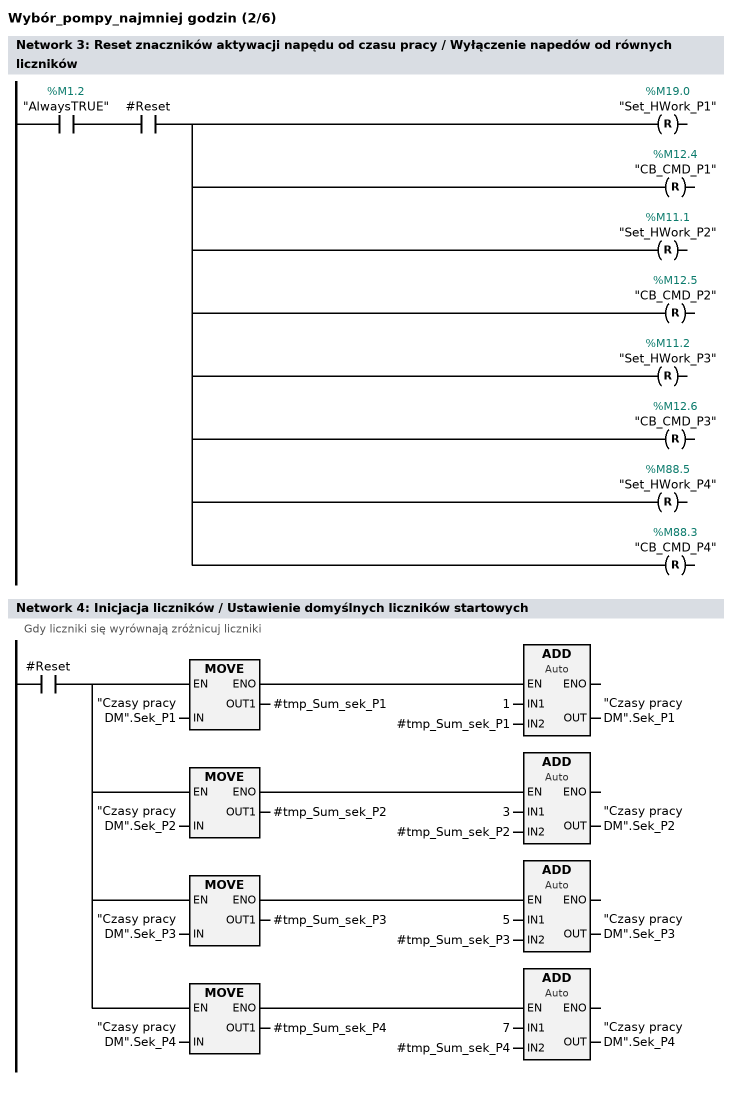
   RUNG wire#powerrail
      Contact( "AlwaysTRUE" )
      Contact( #Reset )
      wire#w1
      R_Coil( "Set_HWork_P1" )
   END_RUNG
   RUNG wire#w1
      R_Coil( "CB_CMD_P1" )
   END_RUNG
   RUNG wire#w1
      R_Coil( "Set_HWork_P2" )
   END_RUNG
   RUNG wire#w1
      R_Coil( "CB_CMD_P2" )
   END_RUNG
   RUNG wire#w1
      R_Coil( "Set_HWork_P3" )
   END_RUNG
   RUNG wire#w1
      R_Coil( "CB_CMD_P3" )
   END_RUNG
   RUNG wire#w1
      R_Coil( "Set_HWork_P4" )
   END_RUNG
   RUNG wire#w1
      R_Coil( "CB_CMD_P4" )
   END_RUNG
   // the same network as SCL:
   IF "AlwaysTRUE" AND #Reset THEN
       "Set_HWork_P1" := FALSE;
       "CB_CMD_P1" := FALSE;
       "Set_HWork_P2" := FALSE;
       "CB_CMD_P2" := FALSE;
       "Set_HWork_P3" := FALSE;
       "CB_CMD_P3" := FALSE;
       "Set_HWork_P4" := FALSE;
       "CB_CMD_P4" := FALSE;
   END_IF;
END_REGION

REGION Network 4: Inicjacja liczników / Ustawienie domyślnych liczników startowych
   // Gdy liczniki się wyrównają zróżnicuj liczniki
   RUNG wire#powerrail
      Contact( #Reset )
      wire#w1
      Move(in := "Czasy pracy DM".Sek_P1, out1 => #tmp_Sum_sek_P1)
      Add(in1 := 1, in2 := #tmp_Sum_sek_P1, out => "Czasy pracy DM".Sek_P1)
   END_RUNG
   RUNG wire#w1
      Move(in := "Czasy pracy DM".Sek_P2, out1 => #tmp_Sum_sek_P2)
      Add(in1 := 3, in2 := #tmp_Sum_sek_P2, out => "Czasy pracy DM".Sek_P2)
   END_RUNG
   RUNG wire#w1
      Move(in := "Czasy pracy DM".Sek_P3, out1 => #tmp_Sum_sek_P3)
      Add(in1 := 5, in2 := #tmp_Sum_sek_P3, out => "Czasy pracy DM".Sek_P3)
   END_RUNG
   RUNG wire#w1
      Move(in := "Czasy pracy DM".Sek_P4, out1 => #tmp_Sum_sek_P4)
      Add(in1 := 7, in2 := #tmp_Sum_sek_P4, out => "Czasy pracy DM".Sek_P4)
   END_RUNG
   // the same network as SCL:
   IF #Reset THEN
       #tmp_Sum_sek_P1 := "Czasy pracy DM".Sek_P1;
       "Czasy pracy DM".Sek_P1 := 1 + #tmp_Sum_sek_P1;
       #tmp_Sum_sek_P2 := "Czasy pracy DM".Sek_P2;
       "Czasy pracy DM".Sek_P2 := 3 + #tmp_Sum_sek_P2;
       #tmp_Sum_sek_P3 := "Czasy pracy DM".Sek_P3;
       "Czasy pracy DM".Sek_P3 := 5 + #tmp_Sum_sek_P3;
       #tmp_Sum_sek_P4 := "Czasy pracy DM".Sek_P4;
       "Czasy pracy DM".Sek_P4 := 7 + #tmp_Sum_sek_P4;
   END_IF;
END_REGION

REGION Network 5: Znacznik wyrównywania czasu pracy z falownika P1 / Znacznik wyrównywania czasu pracy z falownika dla P1
   // %DB10.DBX7.7 - bit tryb automat M7
   // Jesli najmniej godzin pracy to usta znacznik.
   // Ale bierz pod uwagę czy kompresor P2 , P3 już nie pracuje lub nie jest w trybie automat.
   // bit tryb automat P1
   // Jesli najmniej godzin pracy to usta znacznik.
   // Ale bierz po uwagę czy kompresor P1 , P4 już nie pracuje lub nie jest w trybie automat.
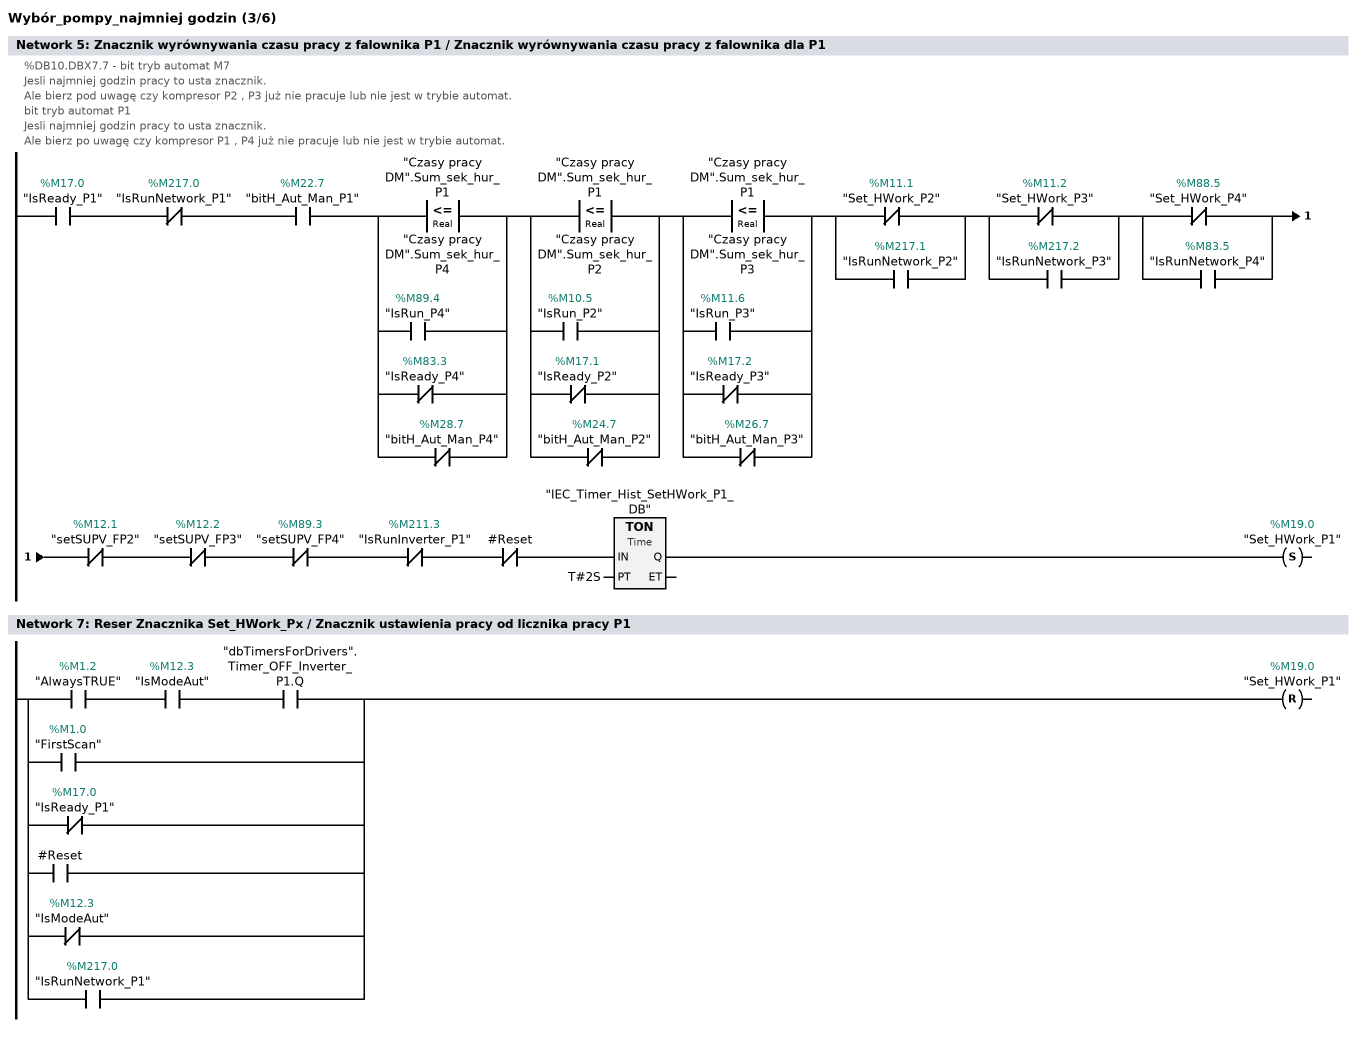
   RUNG wire#powerrail
      Contact( "IsReady_P1" )
      I_Contact( "IsRunNetwork_P1" )
      Contact( "bitH_Aut_Man_P1" )
      wire#w1
      { S7_Templates := "SrcType := Real" } LE_Contact(in1 := "Czasy pracy DM".Sum_sek_hur_P1, in2 := "Czasy pracy DM".Sum_sek_hur_P4)
      wire#w2
      { S7_Templates := "SrcType := Real" } LE_Contact(in1 := "Czasy pracy DM".Sum_sek_hur_P1, in2 := "Czasy pracy DM".Sum_sek_hur_P2)
      wire#w3
      { S7_Templates := "SrcType := Real" } LE_Contact(in1 := "Czasy pracy DM".Sum_sek_hur_P1, in2 := "Czasy pracy DM".Sum_sek_hur_P3)
      wire#w4
      I_Contact( "Set_HWork_P2" )
      wire#w5
      I_Contact( "Set_HWork_P3" )
      wire#w6
      I_Contact( "Set_HWork_P4" )
      wire#w7
      I_Contact( "setSUPV_FP2" )
      I_Contact( "setSUPV_FP3" )
      I_Contact( "setSUPV_FP4" )
      I_Contact( "IsRunInverter_P1" )
      I_Contact( #Reset )
      { S7_Templates := "time_type := Time" } "IEC_Timer_Hist_SetHWork_P1_DB".TON(pt := T#2S, et =>)
      S_Coil( "Set_HWork_P1" )
   END_RUNG
   RUNG wire#w1
      Contact( "IsRun_P4" )
   END_RUNG wire#w2
   RUNG wire#w1
      I_Contact( "IsReady_P4" )
   END_RUNG wire#w2
   RUNG wire#w1
      I_Contact( "bitH_Aut_Man_P4" )
   END_RUNG wire#w2
   RUNG wire#w2
      Contact( "IsRun_P2" )
   END_RUNG wire#w3
   RUNG wire#w2
      I_Contact( "IsReady_P2" )
   END_RUNG wire#w3
   RUNG wire#w2
      I_Contact( "bitH_Aut_Man_P2" )
   END_RUNG wire#w3
   RUNG wire#w3
      Contact( "IsRun_P3" )
   END_RUNG wire#w4
   RUNG wire#w3
      I_Contact( "IsReady_P3" )
   END_RUNG wire#w4
   RUNG wire#w3
      I_Contact( "bitH_Aut_Man_P3" )
   END_RUNG wire#w4
   RUNG wire#w4
      Contact( "IsRunNetwork_P2" )
   END_RUNG wire#w5
   RUNG wire#w5
      Contact( "IsRunNetwork_P3" )
   END_RUNG wire#w6
   RUNG wire#w6
      Contact( "IsRunNetwork_P4" )
   END_RUNG wire#w7
   // the same network as SCL:
   "IEC_Timer_Hist_SetHWork_P1_DB".TON(IN := "IsReady_P1" AND NOT "IsRunNetwork_P1" AND "bitH_Aut_Man_P1" AND (("Czasy pracy DM".Sum_sek_hur_P1 <= "Czasy pracy DM".Sum_sek_hur_P4) OR "IsRun_P4" OR NOT "IsReady_P4" OR NOT "bitH_Aut_Man_P4") AND (("Czasy pracy DM".Sum_sek_hur_P1 <= "Czasy pracy DM".Sum_sek_hur_P2) OR "IsRun_P2" OR NOT "IsReady_P2" OR NOT "bitH_Aut_Man_P2") AND (("Czasy pracy DM".Sum_sek_hur_P1 <= "Czasy pracy DM".Sum_sek_hur_P3) OR "IsRun_P3" OR NOT "IsReady_P3" OR NOT "bitH_Aut_Man_P3") AND (NOT "Set_HWork_P2" OR "IsRunNetwork_P2") AND (NOT "Set_HWork_P3" OR "IsRunNetwork_P3") AND (NOT "Set_HWork_P4" OR "IsRunNetwork_P4") AND NOT "setSUPV_FP2" AND NOT "setSUPV_FP3" AND NOT "setSUPV_FP4" AND NOT "IsRunInverter_P1" AND NOT #Reset,
                           PT := T#2S);
   IF "IEC_Timer_Hist_SetHWork_P1_DB".Q THEN "Set_HWork_P1" := TRUE; END_IF;
END_REGION

REGION Network 6 (SCL): Sprawdzanie czy aktywna w trybie AUT
   IF "Set_HWork_P1" = TRUE AND "bitH_Aut_Man_P1" = FALSE THEN
     // Statement section IF
     "Set_HWork_P1" := FALSE;
     ;
   END_IF;
END_REGION

REGION Network 7: Reser Znacznika Set_HWork_Px / Znacznik ustawienia pracy od licznika pracy P1
   RUNG wire#powerrail
      Contact( "AlwaysTRUE" )
      Contact( "IsModeAut" )
      Contact( "dbTimersForDrivers".Timer_OFF_Inverter_P1.Q )
      wire#w1
      R_Coil( "Set_HWork_P1" )
   END_RUNG
   RUNG wire#powerrail
      Contact( "FirstScan" )
   END_RUNG wire#w1
   RUNG wire#powerrail
      I_Contact( "IsReady_P1" )
   END_RUNG wire#w1
   RUNG wire#powerrail
      Contact( #Reset )
   END_RUNG wire#w1
   RUNG wire#powerrail
      I_Contact( "IsModeAut" )
   END_RUNG wire#w1
   RUNG wire#powerrail
      Contact( "IsRunNetwork_P1" )
   END_RUNG wire#w1
   // the same network as SCL:
   IF ("AlwaysTRUE" AND "IsModeAut" AND "dbTimersForDrivers".Timer_OFF_Inverter_P1.Q) OR "FirstScan" OR NOT "IsReady_P1" OR #Reset OR NOT "IsModeAut" OR "IsRunNetwork_P1" THEN
       "Set_HWork_P1" := FALSE;
   END_IF;
END_REGION

REGION Network 8: Znacznik wyrównywania czasu pracy z falownika P2 / Znacznik wyrównywania czasu pracy z falownika dla P2
   // %DB10.DBX9.7 - bit tryb automat P2
   // Jesli najmniej godzin pracy to usta znacznik.
   // Ale bierz po uwagę czy kompresor P1 , P4 już nie pracuje lub nie jest w trybie automat.
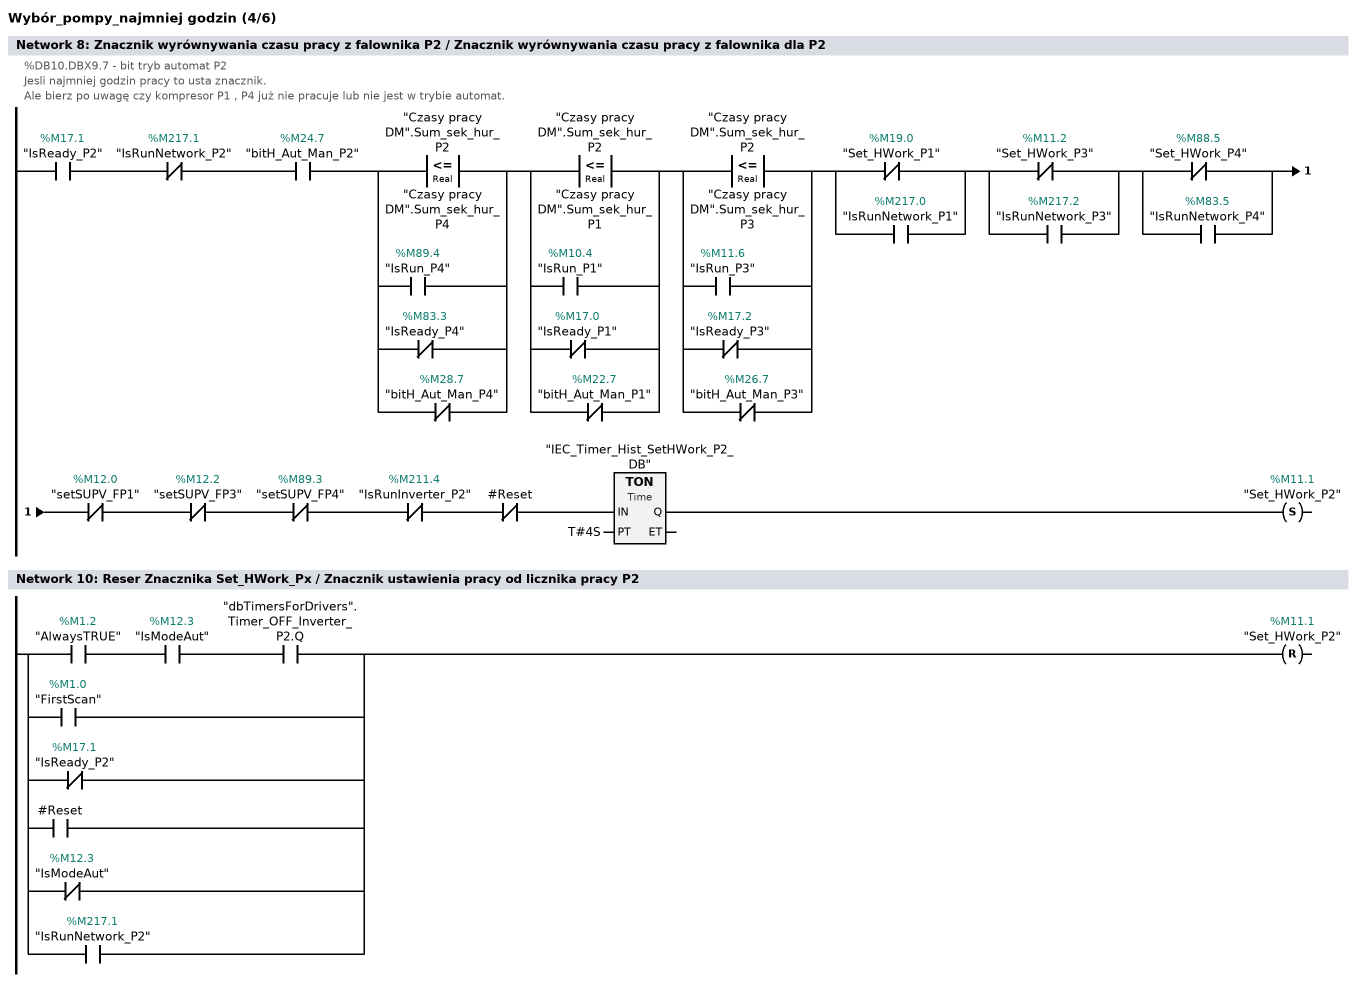
   RUNG wire#powerrail
      Contact( "IsReady_P2" )
      I_Contact( "IsRunNetwork_P2" )
      Contact( "bitH_Aut_Man_P2" )
      wire#w1
      { S7_Templates := "SrcType := Real" } LE_Contact(in1 := "Czasy pracy DM".Sum_sek_hur_P2, in2 := "Czasy pracy DM".Sum_sek_hur_P4)
      wire#w2
      { S7_Templates := "SrcType := Real" } LE_Contact(in1 := "Czasy pracy DM".Sum_sek_hur_P2, in2 := "Czasy pracy DM".Sum_sek_hur_P1)
      wire#w3
      { S7_Templates := "SrcType := Real" } LE_Contact(in1 := "Czasy pracy DM".Sum_sek_hur_P2, in2 := "Czasy pracy DM".Sum_sek_hur_P3)
      wire#w4
      I_Contact( "Set_HWork_P1" )
      wire#w5
      I_Contact( "Set_HWork_P3" )
      wire#w6
      I_Contact( "Set_HWork_P4" )
      wire#w7
      I_Contact( "setSUPV_FP1" )
      I_Contact( "setSUPV_FP3" )
      I_Contact( "setSUPV_FP4" )
      I_Contact( "IsRunInverter_P2" )
      I_Contact( #Reset )
      { S7_Templates := "time_type := Time" } "IEC_Timer_Hist_SetHWork_P2_DB".TON(pt := T#4S, et =>)
      S_Coil( "Set_HWork_P2" )
   END_RUNG
   RUNG wire#w1
      Contact( "IsRun_P4" )
   END_RUNG wire#w2
   RUNG wire#w1
      I_Contact( "IsReady_P4" )
   END_RUNG wire#w2
   RUNG wire#w1
      I_Contact( "bitH_Aut_Man_P4" )
   END_RUNG wire#w2
   RUNG wire#w2
      Contact( "IsRun_P1" )
   END_RUNG wire#w3
   RUNG wire#w2
      I_Contact( "IsReady_P1" )
   END_RUNG wire#w3
   RUNG wire#w2
      I_Contact( "bitH_Aut_Man_P1" )
   END_RUNG wire#w3
   RUNG wire#w3
      Contact( "IsRun_P3" )
   END_RUNG wire#w4
   RUNG wire#w3
      I_Contact( "IsReady_P3" )
   END_RUNG wire#w4
   RUNG wire#w3
      I_Contact( "bitH_Aut_Man_P3" )
   END_RUNG wire#w4
   RUNG wire#w4
      Contact( "IsRunNetwork_P1" )
   END_RUNG wire#w5
   RUNG wire#w5
      Contact( "IsRunNetwork_P3" )
   END_RUNG wire#w6
   RUNG wire#w6
      Contact( "IsRunNetwork_P4" )
   END_RUNG wire#w7
   // the same network as SCL:
   "IEC_Timer_Hist_SetHWork_P2_DB".TON(IN := "IsReady_P2" AND NOT "IsRunNetwork_P2" AND "bitH_Aut_Man_P2" AND (("Czasy pracy DM".Sum_sek_hur_P2 <= "Czasy pracy DM".Sum_sek_hur_P4) OR "IsRun_P4" OR NOT "IsReady_P4" OR NOT "bitH_Aut_Man_P4") AND (("Czasy pracy DM".Sum_sek_hur_P2 <= "Czasy pracy DM".Sum_sek_hur_P1) OR "IsRun_P1" OR NOT "IsReady_P1" OR NOT "bitH_Aut_Man_P1") AND (("Czasy pracy DM".Sum_sek_hur_P2 <= "Czasy pracy DM".Sum_sek_hur_P3) OR "IsRun_P3" OR NOT "IsReady_P3" OR NOT "bitH_Aut_Man_P3") AND (NOT "Set_HWork_P1" OR "IsRunNetwork_P1") AND (NOT "Set_HWork_P3" OR "IsRunNetwork_P3") AND (NOT "Set_HWork_P4" OR "IsRunNetwork_P4") AND NOT "setSUPV_FP1" AND NOT "setSUPV_FP3" AND NOT "setSUPV_FP4" AND NOT "IsRunInverter_P2" AND NOT #Reset,
                           PT := T#4S);
   IF "IEC_Timer_Hist_SetHWork_P2_DB".Q THEN "Set_HWork_P2" := TRUE; END_IF;
END_REGION

REGION Network 9 (SCL): Sprawdzanie czy aktywna w trybie AUT
   IF "Set_HWork_P2" = TRUE AND "bitH_Aut_Man_P2" = FALSE THEN
     // Statement section IF
     "Set_HWork_P2" := FALSE;
     ;
   END_IF;
END_REGION

REGION Network 10: Reser Znacznika Set_HWork_Px / Znacznik ustawienia pracy od licznika pracy P2
   RUNG wire#powerrail
      Contact( "AlwaysTRUE" )
      Contact( "IsModeAut" )
      Contact( "dbTimersForDrivers".Timer_OFF_Inverter_P2.Q )
      wire#w1
      R_Coil( "Set_HWork_P2" )
   END_RUNG
   RUNG wire#powerrail
      Contact( "FirstScan" )
   END_RUNG wire#w1
   RUNG wire#powerrail
      I_Contact( "IsReady_P2" )
   END_RUNG wire#w1
   RUNG wire#powerrail
      Contact( #Reset )
   END_RUNG wire#w1
   RUNG wire#powerrail
      I_Contact( "IsModeAut" )
   END_RUNG wire#w1
   RUNG wire#powerrail
      Contact( "IsRunNetwork_P2" )
   END_RUNG wire#w1
   // the same network as SCL:
   IF ("AlwaysTRUE" AND "IsModeAut" AND "dbTimersForDrivers".Timer_OFF_Inverter_P2.Q) OR "FirstScan" OR NOT "IsReady_P2" OR #Reset OR NOT "IsModeAut" OR "IsRunNetwork_P2" THEN
       "Set_HWork_P2" := FALSE;
   END_IF;
END_REGION

REGION Network 11: Znacznik wyrównywania czasu pracy z falownika P3 / Znacznik wyrównywania czasu pracy z falownika P3
   // bit tryb automat P3
   // Jesli najmniej godzin pracy to usta znacznik.
   // Ale bierz po uwagę czy P1, P4 już nie pracuje lub nie jest w trybie automat.
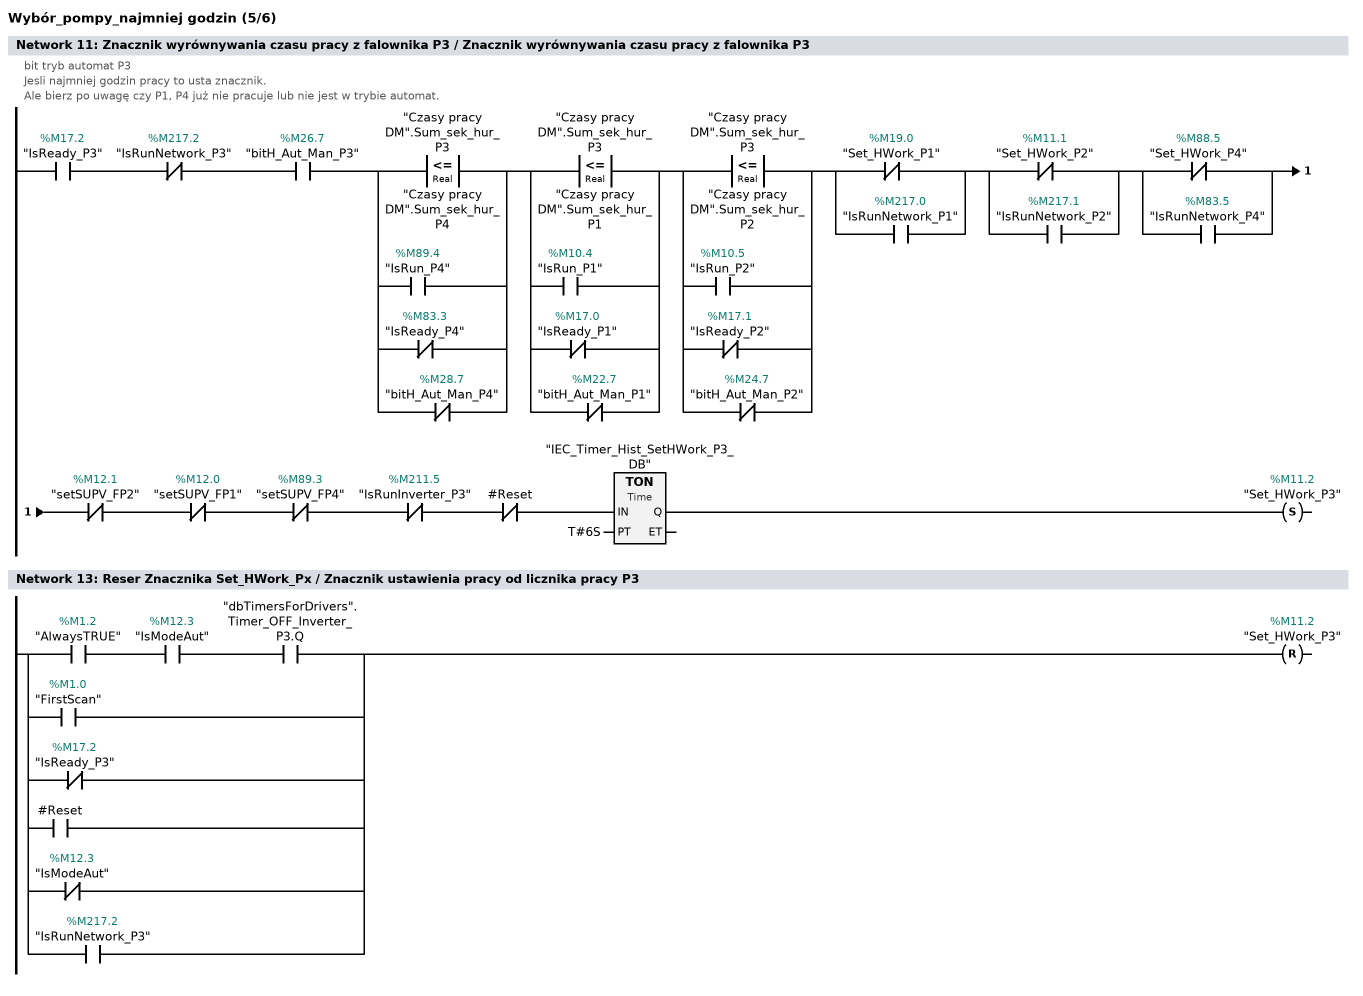
   RUNG wire#powerrail
      Contact( "IsReady_P3" )
      I_Contact( "IsRunNetwork_P3" )
      Contact( "bitH_Aut_Man_P3" )
      wire#w1
      { S7_Templates := "SrcType := Real" } LE_Contact(in1 := "Czasy pracy DM".Sum_sek_hur_P3, in2 := "Czasy pracy DM".Sum_sek_hur_P4)
      wire#w2
      { S7_Templates := "SrcType := Real" } LE_Contact(in1 := "Czasy pracy DM".Sum_sek_hur_P3, in2 := "Czasy pracy DM".Sum_sek_hur_P1)
      wire#w3
      { S7_Templates := "SrcType := Real" } LE_Contact(in1 := "Czasy pracy DM".Sum_sek_hur_P3, in2 := "Czasy pracy DM".Sum_sek_hur_P2)
      wire#w4
      I_Contact( "Set_HWork_P1" )
      wire#w5
      I_Contact( "Set_HWork_P2" )
      wire#w6
      I_Contact( "Set_HWork_P4" )
      wire#w7
      I_Contact( "setSUPV_FP2" )
      I_Contact( "setSUPV_FP1" )
      I_Contact( "setSUPV_FP4" )
      I_Contact( "IsRunInverter_P3" )
      I_Contact( #Reset )
      { S7_Templates := "time_type := Time" } "IEC_Timer_Hist_SetHWork_P3_DB".TON(pt := T#6S, et =>)
      S_Coil( "Set_HWork_P3" )
   END_RUNG
   RUNG wire#w1
      Contact( "IsRun_P4" )
   END_RUNG wire#w2
   RUNG wire#w1
      I_Contact( "IsReady_P4" )
   END_RUNG wire#w2
   RUNG wire#w1
      I_Contact( "bitH_Aut_Man_P4" )
   END_RUNG wire#w2
   RUNG wire#w2
      Contact( "IsRun_P1" )
   END_RUNG wire#w3
   RUNG wire#w2
      I_Contact( "IsReady_P1" )
   END_RUNG wire#w3
   RUNG wire#w2
      I_Contact( "bitH_Aut_Man_P1" )
   END_RUNG wire#w3
   RUNG wire#w3
      Contact( "IsRun_P2" )
   END_RUNG wire#w4
   RUNG wire#w3
      I_Contact( "IsReady_P2" )
   END_RUNG wire#w4
   RUNG wire#w3
      I_Contact( "bitH_Aut_Man_P2" )
   END_RUNG wire#w4
   RUNG wire#w4
      Contact( "IsRunNetwork_P1" )
   END_RUNG wire#w5
   RUNG wire#w5
      Contact( "IsRunNetwork_P2" )
   END_RUNG wire#w6
   RUNG wire#w6
      Contact( "IsRunNetwork_P4" )
   END_RUNG wire#w7
   // the same network as SCL:
   "IEC_Timer_Hist_SetHWork_P3_DB".TON(IN := "IsReady_P3" AND NOT "IsRunNetwork_P3" AND "bitH_Aut_Man_P3" AND (("Czasy pracy DM".Sum_sek_hur_P3 <= "Czasy pracy DM".Sum_sek_hur_P4) OR "IsRun_P4" OR NOT "IsReady_P4" OR NOT "bitH_Aut_Man_P4") AND (("Czasy pracy DM".Sum_sek_hur_P3 <= "Czasy pracy DM".Sum_sek_hur_P1) OR "IsRun_P1" OR NOT "IsReady_P1" OR NOT "bitH_Aut_Man_P1") AND (("Czasy pracy DM".Sum_sek_hur_P3 <= "Czasy pracy DM".Sum_sek_hur_P2) OR "IsRun_P2" OR NOT "IsReady_P2" OR NOT "bitH_Aut_Man_P2") AND (NOT "Set_HWork_P1" OR "IsRunNetwork_P1") AND (NOT "Set_HWork_P2" OR "IsRunNetwork_P2") AND (NOT "Set_HWork_P4" OR "IsRunNetwork_P4") AND NOT "setSUPV_FP2" AND NOT "setSUPV_FP1" AND NOT "setSUPV_FP4" AND NOT "IsRunInverter_P3" AND NOT #Reset,
                           PT := T#6S);
   IF "IEC_Timer_Hist_SetHWork_P3_DB".Q THEN "Set_HWork_P3" := TRUE; END_IF;
END_REGION

REGION Network 12 (SCL): Sprawdzanie czy aktywna w trybie AUT
   IF "Set_HWork_P3" = TRUE AND "bitH_Aut_Man_P3" = FALSE THEN
     // Statement section IF
     "Set_HWork_P3" := FALSE;
     ;
   END_IF;
END_REGION

REGION Network 13: Reser Znacznika Set_HWork_Px / Znacznik ustawienia pracy od licznika pracy P3
   RUNG wire#powerrail
      Contact( "AlwaysTRUE" )
      Contact( "IsModeAut" )
      Contact( "dbTimersForDrivers".Timer_OFF_Inverter_P3.Q )
      wire#w1
      R_Coil( "Set_HWork_P3" )
   END_RUNG
   RUNG wire#powerrail
      Contact( "FirstScan" )
   END_RUNG wire#w1
   RUNG wire#powerrail
      I_Contact( "IsReady_P3" )
   END_RUNG wire#w1
   RUNG wire#powerrail
      Contact( #Reset )
   END_RUNG wire#w1
   RUNG wire#powerrail
      I_Contact( "IsModeAut" )
   END_RUNG wire#w1
   RUNG wire#powerrail
      Contact( "IsRunNetwork_P3" )
   END_RUNG wire#w1
   // the same network as SCL:
   IF ("AlwaysTRUE" AND "IsModeAut" AND "dbTimersForDrivers".Timer_OFF_Inverter_P3.Q) OR "FirstScan" OR NOT "IsReady_P3" OR #Reset OR NOT "IsModeAut" OR "IsRunNetwork_P3" THEN
       "Set_HWork_P3" := FALSE;
   END_IF;
END_REGION

REGION Network 14: Znacznik wyrównywania czasu pracy z falownika P4 / Znacznik wyrównywania czasu pracy z falownika P4
   // bit tryb automat P4
   // Jesli najmniej godzin pracy to usta znacznik.
   // Ale bierz po uwagę czy P1, P4 już nie pracuje lub nie jest w trybie automat.
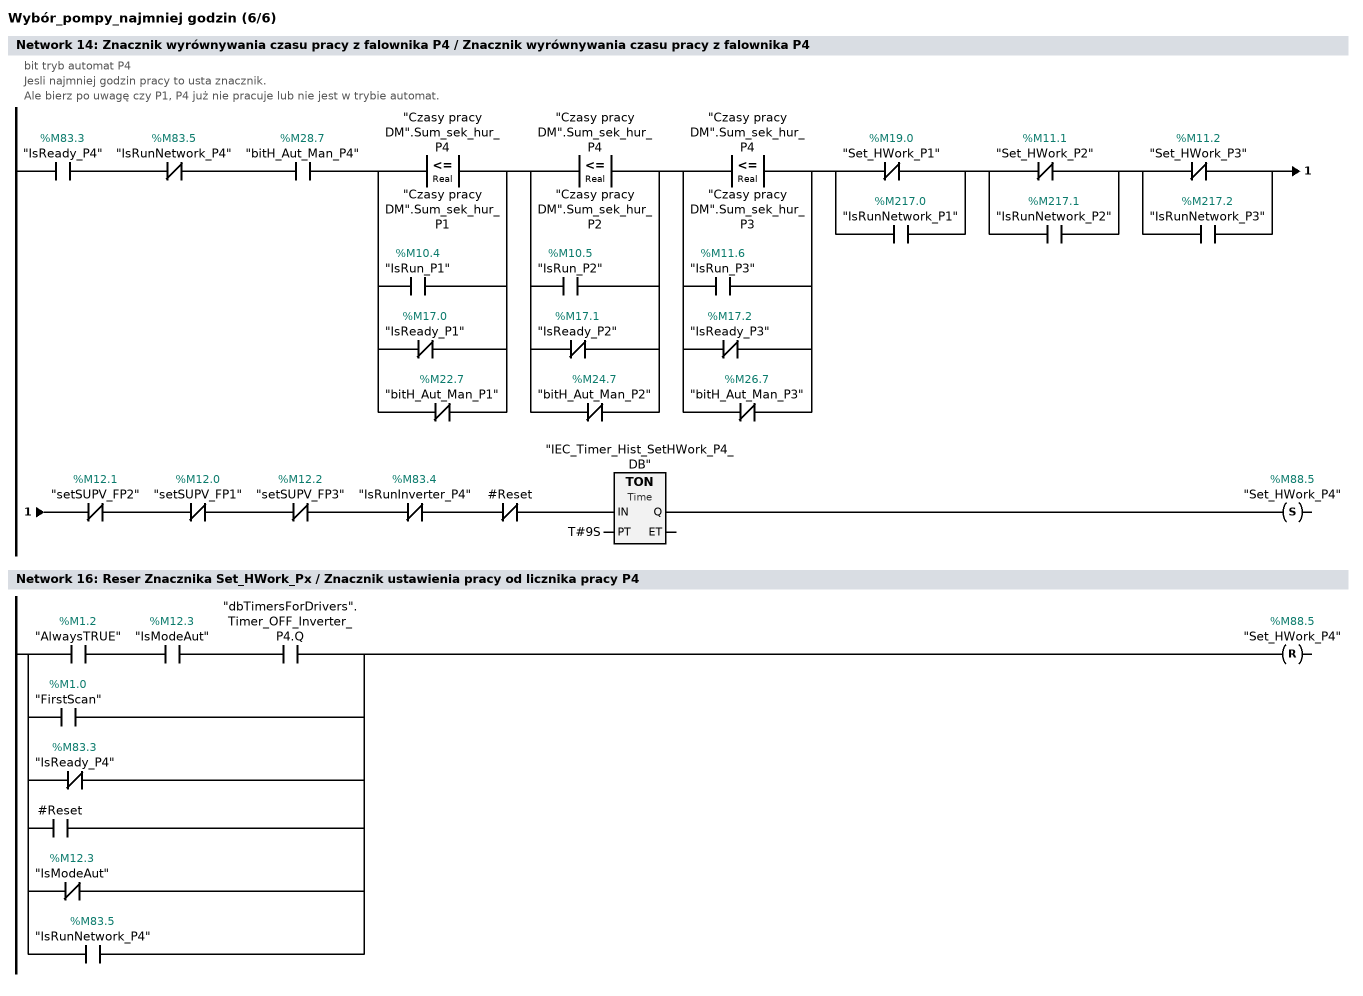
   RUNG wire#powerrail
      Contact( "IsReady_P4" )
      I_Contact( "IsRunNetwork_P4" )
      Contact( "bitH_Aut_Man_P4" )
      wire#w1
      { S7_Templates := "SrcType := Real" } LE_Contact(in1 := "Czasy pracy DM".Sum_sek_hur_P4, in2 := "Czasy pracy DM".Sum_sek_hur_P1)
      wire#w2
      { S7_Templates := "SrcType := Real" } LE_Contact(in1 := "Czasy pracy DM".Sum_sek_hur_P4, in2 := "Czasy pracy DM".Sum_sek_hur_P2)
      wire#w3
      { S7_Templates := "SrcType := Real" } LE_Contact(in1 := "Czasy pracy DM".Sum_sek_hur_P4, in2 := "Czasy pracy DM".Sum_sek_hur_P3)
      wire#w4
      I_Contact( "Set_HWork_P1" )
      wire#w5
      I_Contact( "Set_HWork_P2" )
      wire#w6
      I_Contact( "Set_HWork_P3" )
      wire#w7
      I_Contact( "setSUPV_FP2" )
      I_Contact( "setSUPV_FP1" )
      I_Contact( "setSUPV_FP3" )
      I_Contact( "IsRunInverter_P4" )
      I_Contact( #Reset )
      { S7_Templates := "time_type := Time" } "IEC_Timer_Hist_SetHWork_P4_DB".TON(pt := T#9S, et =>)
      S_Coil( "Set_HWork_P4" )
   END_RUNG
   RUNG wire#w1
      Contact( "IsRun_P1" )
   END_RUNG wire#w2
   RUNG wire#w1
      I_Contact( "IsReady_P1" )
   END_RUNG wire#w2
   RUNG wire#w1
      I_Contact( "bitH_Aut_Man_P1" )
   END_RUNG wire#w2
   RUNG wire#w2
      Contact( "IsRun_P2" )
   END_RUNG wire#w3
   RUNG wire#w2
      I_Contact( "IsReady_P2" )
   END_RUNG wire#w3
   RUNG wire#w2
      I_Contact( "bitH_Aut_Man_P2" )
   END_RUNG wire#w3
   RUNG wire#w3
      Contact( "IsRun_P3" )
   END_RUNG wire#w4
   RUNG wire#w3
      I_Contact( "IsReady_P3" )
   END_RUNG wire#w4
   RUNG wire#w3
      I_Contact( "bitH_Aut_Man_P3" )
   END_RUNG wire#w4
   RUNG wire#w4
      Contact( "IsRunNetwork_P1" )
   END_RUNG wire#w5
   RUNG wire#w5
      Contact( "IsRunNetwork_P2" )
   END_RUNG wire#w6
   RUNG wire#w6
      Contact( "IsRunNetwork_P3" )
   END_RUNG wire#w7
   // the same network as SCL:
   "IEC_Timer_Hist_SetHWork_P4_DB".TON(IN := "IsReady_P4" AND NOT "IsRunNetwork_P4" AND "bitH_Aut_Man_P4" AND (("Czasy pracy DM".Sum_sek_hur_P4 <= "Czasy pracy DM".Sum_sek_hur_P1) OR "IsRun_P1" OR NOT "IsReady_P1" OR NOT "bitH_Aut_Man_P1") AND (("Czasy pracy DM".Sum_sek_hur_P4 <= "Czasy pracy DM".Sum_sek_hur_P2) OR "IsRun_P2" OR NOT "IsReady_P2" OR NOT "bitH_Aut_Man_P2") AND (("Czasy pracy DM".Sum_sek_hur_P4 <= "Czasy pracy DM".Sum_sek_hur_P3) OR "IsRun_P3" OR NOT "IsReady_P3" OR NOT "bitH_Aut_Man_P3") AND (NOT "Set_HWork_P1" OR "IsRunNetwork_P1") AND (NOT "Set_HWork_P2" OR "IsRunNetwork_P2") AND (NOT "Set_HWork_P3" OR "IsRunNetwork_P3") AND NOT "setSUPV_FP2" AND NOT "setSUPV_FP1" AND NOT "setSUPV_FP3" AND NOT "IsRunInverter_P4" AND NOT #Reset,
                           PT := T#9S);
   IF "IEC_Timer_Hist_SetHWork_P4_DB".Q THEN "Set_HWork_P4" := TRUE; END_IF;
END_REGION

REGION Network 15 (SCL): Sprawdzanie czy aktywna w trybie AUT
   IF "Set_HWork_P4" = TRUE AND "bitH_Aut_Man_P4" = FALSE THEN
     // Statement section IF
     "Set_HWork_P4" := FALSE;
     ;
   END_IF;
END_REGION

REGION Network 16: Reser Znacznika Set_HWork_Px / Znacznik ustawienia pracy od licznika pracy P4
   RUNG wire#powerrail
      Contact( "AlwaysTRUE" )
      Contact( "IsModeAut" )
      Contact( "dbTimersForDrivers".Timer_OFF_Inverter_P4.Q )
      wire#w1
      R_Coil( "Set_HWork_P4" )
   END_RUNG
   RUNG wire#powerrail
      Contact( "FirstScan" )
   END_RUNG wire#w1
   RUNG wire#powerrail
      I_Contact( "IsReady_P4" )
   END_RUNG wire#w1
   RUNG wire#powerrail
      Contact( #Reset )
   END_RUNG wire#w1
   RUNG wire#powerrail
      I_Contact( "IsModeAut" )
   END_RUNG wire#w1
   RUNG wire#powerrail
      Contact( "IsRunNetwork_P4" )
   END_RUNG wire#w1
   // the same network as SCL:
   IF ("AlwaysTRUE" AND "IsModeAut" AND "dbTimersForDrivers".Timer_OFF_Inverter_P4.Q) OR "FirstScan" OR NOT "IsReady_P4" OR #Reset OR NOT "IsModeAut" OR "IsRunNetwork_P4" THEN
       "Set_HWork_P4" := FALSE;
   END_IF;
END_REGION
END_FUNCTION

FUNCTION "ClearError_Modbus" : Void
{ S7_Optimized_Access := 'TRUE' }
AUTHOR : rtecmer
VERSION : 0.1
   VAR_TEMP 
      set_error_RTU : Bool;
   END_VAR


BEGIN
	
	(*
	//=============================================================================
	//(JZWiK S.A Radosław Tecmer)
	//(c)Copyright (2021) All Rights Reserved
	//-----------------------------------------------------------------------------
	//Testowane z:   (system docelowy z  FW 4.4)
	//Pakiet inżynierski:   TIA Portal (V14 Sp1 Update 9)
	//Ograniczenia:  ( - )
	//Wymagania:  (minimalne S7-1200 CPU 1215C FW 4.2 .)
	//Funkcjonalnośc: (Obsługa błedów na magistrali Modbus RTU, inicjacja pętli po konfliktach )
	//-----------------------------------------------------------------------------
	//Zmainy wprowadzone:
	//Wersja  Data       Osoba wprowadzająca zmiany - ekspert
	//01.00.00 17.11.2021 (Tecmer Radosław - twórca) Pieresza wersja 01.00.00
	//=============================================================================
	*)
	
	REGION Główny błąd - wszystkie pętle nie działają
	  //kasowanie wartości zmiennych errorStatus odblokowanie magistrali
	  IF "setErrorModbsmasterMPP04_1" AND "setErrorModbsmasterFal" THEN
	    //ustaw znacznik błędu
	    "db10organizacyjna".setRTU_Error := TRUE;
	    // resetuj mdbusMastererror dla wszystkich pętli
	    "dbTags_master_Fal_1".modbusMaster.error := FALSE;
	    "dbTags_master_MPP04_1".modbusMaster.error := FALSE;
	    
	  ELSE
	    "db10organizacyjna".setRTU_Error := FALSE;
	    ;
	  END_IF;
	  
	END_REGION
	
	IF ("db10organizacyjna".RTU_Fal_1errorStatus = 0) AND ("db10organizacyjna".RTU_MPP04_1errorStatus = 0) THEN
	  // kasowanie znacznika błędu komunikacj modbus rtu
	  "db10organizacyjna".setRTU_Error := FALSE;
	  ;
	END_IF;
	
	
	
	
	
	REGION Falownik Modbau RTU
	  // Sprawdzanie czy 
	  IF "dbTags_master_Fal_1".step = 27 THEN
	    // Statement section IF
	    "dbTags_master_Fal_1".modbusMaster.error := FALSE;
	    "dbTags_master_Fal_1".modbusMaster.busy := FALSE;
	    "dbTags_master_Fal_1".modbusMaster.status:= 0;
	    
	   
	   // jeśli MPP04_1 kod błedu 80C8 (brak urządzenia na linni) to uruchom pętlę modbus dla falownika
	    IF "dbTags_master_MPP04_1".modbusMaster.status = 16#80C8 AND ("dbTags_master_Fal_1".step = 27 OR "dbTags_master_Fal_1".step = 25 )
	    THEN
	      // Statement section 
	      "setErrorModbsmasterFal" := FALSE;
	      "dbTags_master_Fal_1".step := 1;
	      
	      ;
	    END_IF;
	    
	    ;
	  END_IF;
	  
	  // awaria komunikacji z falownikiem Modbus-RTU
	  IF "setErrorModbsmasterFal" THEN
	    // ustaw bit awarii 
	    "dbzarządzanie".sterowanie_1.awaria_modbus_falownik:= TRUE
	    ;
	  END_IF;
	  
	  // kasowanie biti awarii komunikacji falownika Modbus-RTU
	  IF "memStep_errorFal" = 100 THEN
	    // kasowanie
	    "dbzarządzanie".sterowanie_1.awaria_modbus_falownik:= FALSE
	    ;
	  END_IF;
	  
	  
	END_REGION
	
	REGION MPP04-1 Modbau RTU
	  // Sprawdzanie czy 
	  IF "dbTags_master_MPP04_1".step = 27 AND "dbTags_master_Fal_1".step = 27
	     THEN
	    // 
	    "dbTags_master_MPP04_1".modbusMaster.error := FALSE;
	    "dbTags_master_MPP04_1".modbusMaster.busy := FALSE;
	    "dbTags_master_MPP04_1".modbusMaster.status := 0;
	    "dbTags_master_Fal_1".step := 1;
	    
	    ;
	  END_IF;
	  
	  IF "dbTags_master_MPP04_1".step = 27
	  THEN
	    // 
	    "dbTags_master_MPP04_1".modbusMaster.error := FALSE;
	    "dbTags_master_MPP04_1".modbusMaster.busy := FALSE;
	    "dbTags_master_MPP04_1".modbusMaster.status := 0;
	    //"dbTags_master_MPP04_1".step := 25;
	    
	    ;
	  END_IF;
	  
	  
	  // awaria komunikacji z MPO04 Modbus-RTU
	  IF "setErrorModbsmasterMPP04_1"  THEN
	    // ustaw bit awarii po czasie zwłoki 
	    "IEC_Timer_errorRTU_histereza_DB".TON(IN:="setErrorModbsmasterMPP04_1",
	                                          PT:=T#30S);
	    #set_error_RTU := "IEC_Timer_errorRTU_histereza_DB".Q;
	    "dbzarządzanie".sterowanie_1.awaria_modbus_przepływ_pomp := #set_error_RTU;
	  ELSE
	    #set_error_RTU := FALSE;
	    ;
	  END_IF;
	  
	  // kasowanie biti awarii komunikacjiModbus-RTU
	  IF "memStep_errorMPP04-1" = 100  AND "setErrorModbsmasterMPP04_1" = FALSE THEN
	    // kasowanie
	    "dbzarządzanie".sterowanie_1.awaria_modbus_przepływ_pomp:= FALSE
	    ;
	  END_IF;
	  
	END_REGION
	
	
	
	//Modbus RTU Error Code RESET
	REGION Modbus RTU Error Code
	  // Ustaw reset modbus rtu
	  IF "db10organizacyjna".RTU_stepRESET THEN
	    // Ustawienie domyślnych satrtowych 
	    "dbTags_master_MPP04_1".step := 1;
	    
	    "dbTags_master_Fal_1".step := 25;
	    "dbTags_slave_RTU".step := 25;
	    
	    // Zerowanie kodu błędu
	    "dbTags_master_MPP04_1".modbusMaster.errorStatus := 0;
	    "dbTags_slave_RTU".modbusMaster.errorStatus := 0;
	    
	    "db10organizacyjna".RTU_stepRESET := 0;
	    ;
	  END_IF;
	  
	  
	END_REGION
	
	// Ustawienie Błędu Modbus RTU 
	REGION Set Fault Modbus RTU 
	  // Jeśli zmienna kodu błędu różna od 0 to ustaw znacznik błędu Modbus w bloku danych SCADA
	  // i przekaż wartość błędów
	  IF "dbzarządzanie".sterowanie_1."alarm-modbus" = TRUE
	    
	  THEN
	    
	    "db10organizacyjna".RTU_MPP04_1errorStatus := "dbTags_master_MPP04_1".modbusMaster.errorStatus;
	    // Trzeba dopisać przekazanie błędu z PLC Zasuwy
	   // "DB10_instance_SCADA".RTU_MPP04_2errorStatus := "dbTags_master_MPP04_2".modbusMaster.errorStatus;
	    "db10organizacyjna".RTU_Fal_1errorStatus := "dbTags_master_Fal_1".modbusMaster.errorStatus;
	    "db10organizacyjna".RTU_MT101 := "dbTags_slave_RTU".modbusMaster.errorStatus;
	  ELSE
	    //
	    ;
	    ;
	  END_IF;
	  
	  
	  // Modbus przekaż bit do instancji SCADA Alarm ostrzeżenie kłoport z Modbau
	  // Przynajmniej jeden slave nie odpowiada
	  IF "dbTags_master_Fal_1".step = 27 OR "dbTags_master_MPP04_1".step = 27 
	 
	  THEN
	    "dbzarządzanie".sterowanie_1."alarm-warning" := TRUE;
	
	    ;
	    
	  END_IF;
	  
	  IF "db10organizacyjna".RTU_Fal_1errorStatus = 0 AND "db10organizacyjna".RTU_MPP04_1errorStatus = 0 THEN
	  // kasuj ostrzeżenie
	    "dbzarządzanie".sterowanie_1."alarm-warning" := FALSE;
	    ;
	  ;
	END_IF;
	
	  
	  
	  
	  
	END_REGION
	
	
	
	
	
END_FUNCTION

FUNCTION_BLOCK "Alarm_min_magistrala_B5"
TITLE = Start procedury awarujnego pompowania
{ S7_Optimized_Access := 'TRUE' }
AUTHOR : rt69
VERSION : 0.1
//Funkcja rozpoczyna procedurę awaryjnego sterowaia zasilaniem na magistralę 
   VAR_OUTPUT 
      bit_alarm_magistrala_min { ExternalAccessible := 'False'; ExternalVisible := 'False'; ExternalWritable := 'False'} : Bool := false;   // bit alarmmagistrala awaria niskie ciśnienie
   END_VAR

   VAR_IN_OUT 
      bit_off_alarm_niskie_magistrala { ExternalAccessible := 'False'; ExternalVisible := 'False'; ExternalWritable := 'False'} : Bool;   // bit koniec alarmu niskie bar magistrala
      "tempStrategia Pompownia" : Int := 16#0;   // przechwycone słowo strategii pompownia
      "actStrategia Pompownia" : Int;   // Słowo reprezentujące strategie sterowania pompownią (wyłączona , przetłaczanie , dosilanie,automat)
   END_VAR

   VAR 
      memTriger_Strategia { ExternalAccessible := 'False'; ExternalVisible := 'False'; ExternalWritable := 'False'} : Bool;   // pamięć zbocza
      bit_normalne_magistrala { ExternalAccessible := 'False'; ExternalVisible := 'False'; ExternalWritable := 'False'} : Bool;   // bit detekcjinormalnego cisnienia magistrala
      bit_niskie_magistrala { ExternalAccessible := 'False'; ExternalVisible := 'False'; ExternalWritable := 'False'} : Bool;   // bit detekcji niskiego cisnienia magistrala
   END_VAR


BEGIN
	(*
	//=============================================================================
	//(JZWiK S.A Radosław Tecmer)
	//(c)Copyright (2021) All Rights Reserved
	//-----------------------------------------------------------------------------
	//Testowane z:   (system docelowy z  FW 4.4)
	//Pakiet inżynierski:   TIA Portal (V14 Sp1 Update 9)
	//Ograniczenia:  ( - )
	//Wymagania:  (minimalne S7-1200 CPU 1215C FW 4.2 .)
	//Funkcjonalnośc: (kontrola cisnienia magistrali, sterowanie strategią gdy 
	                    awaria ciśnienia B5 i powrót poprawnego)
	//-----------------------------------------------------------------------------
	//Zmainy wprowadzone:
	//Wersja  Data       Osoba wprowadzająca zmiany - ekspert
	//01.00.00 17.11.2021 (Tecmer Radosław - twórca) Pieresza wersja 01.00.00
	//=============================================================================
	*)
	
	
	
	REGION Kontrola  cięnieia magistrali, alarm niskie magistrala czujnik B5
	  
	  // Kontrola ciśnienia zasilania z magistrali B5
	  // Detekcja zaistnienia awarii zasilania na magistrali
	  IF "dbdane".Act_Value_B5_magistrala_bar < "dbHold_RRG".Sending.set_magistrala_alarm_min_bar THEN
	    // Ustaw bit za niskie ciśnienie
	    #bit_niskie_magistrala := TRUE;
	  ELSE
	    
	    ;
	  END_IF;
	  
	  "R_TRIG_DB_przechwycenie_strategii"(CLK := #bit_niskie_magistrala,
	                                      Q => #memTriger_Strategia);
	  IF #memTriger_Strategia THEN
	    // zatrzaśniecie przechwyconą strategię 
	    #"tempStrategia Pompownia" := #"actStrategia Pompownia";
	    IF #"tempStrategia Pompownia" = 0 THEN
	      // to wpisz domyślną 2
	      #"tempStrategia Pompownia" := 2;
	      ;
	    END_IF;
	    
	    ;
	  END_IF;
	  
	  // Histereza na ustawienie alarmu "niskie ćiśnienie na magistrali"
	  "IEC_Timer_AlarmMagistrala_Niskie_DB".TON(IN := #bit_niskie_magistrala,
	                                            PT := T#14M,
	                                            Q => #bit_alarm_magistrala_min);
	  
	  
	  
	  // Sprawdzanie powrotu zasilania z magistrali czujnik B5
	  IF "dbdane".Act_Value_B5_magistrala_bar > 7.4 THEN
	    // Ustaw bit za normalne ciśnienie
	    #bit_normalne_magistrala := TRUE;
	    
	  ELSE
	    #bit_normalne_magistrala := FALSE;
	    ;
	  END_IF;
	  
	  //Histerez na powrót normalnego zasilania z magistrali
	  "IEC_Timer_resetAlarmMagistrala_Niskie_DB".TON(IN := #bit_normalne_magistrala,
	                                                 Q => #bit_off_alarm_niskie_magistrala,
	                                                 PT := T#4M);
	  
	  IF #bit_off_alarm_niskie_magistrala THEN
	    // kasuj alarm niskie magistrala
	    #bit_niskie_magistrala := FALSE;
	    ;
	  END_IF;
	  
	END_REGION
END_FUNCTION_BLOCK

FUNCTION_BLOCK "Strategia sterowaia Z11"
TITLE = Strategia sterowania 
{ S7_Optimized_Access := 'TRUE' }
AUTHOR : rtecmer
VERSION : 0.1
//Funkcja sterowania przełączaniem kieunku pompowania Z11 - przetłaczania kierunek miasto, Z12 - dosilanie w kierunku magistrali
   VAR_INPUT 
      bit_alarm_magistrala_min { ExternalAccessible := 'False'; ExternalVisible := 'False'; ExternalWritable := 'False'} : Bool := false;   // bit alarmmagistrala awaria niskie ciśnienie
   END_VAR

   VAR_IN_OUT 
      CMD_Open_Z11 : Bool;   // znacznik sterowania otwieraniem
      CMD_Close_Z11 : Bool;   // znacznik sterowania otwieraniem
   END_VAR

   VAR 
      bit_set_open_Z11 { ExternalAccessible := 'False'; ExternalVisible := 'False'; ExternalWritable := 'False'} : Bool;   // bit inicjacji otwierania zasuwy w trybie strategii
      bit_set_open_Z12 { ExternalAccessible := 'False'; ExternalVisible := 'False'; ExternalWritable := 'False'} : Bool;   // bit inicjacji otwierania zasuwy w trybie strategii
      bit_hist_open_Z11 { ExternalAccessible := 'False'; ExternalVisible := 'False'; ExternalWritable := 'False'} : Bool;   // bit opóźnienia reakcji
      bit_hist_open_Z12 { ExternalAccessible := 'False'; ExternalVisible := 'False'; ExternalWritable := 'False'} : Bool;   // bit opóźnienia reakcji
      bit_set_close_Z11 { ExternalAccessible := 'False'; ExternalVisible := 'False'; ExternalWritable := 'False'} : Bool;   // bit inicjacji otwierania zasuwy w trybie strategii
      bit_set_close_Z12 { ExternalAccessible := 'False'; ExternalVisible := 'False'; ExternalWritable := 'False'} : Bool;   // bit inicjacji otwierania zasuwy w trybie strategii
      bit_hist_close_Z11 { ExternalAccessible := 'False'; ExternalVisible := 'False'; ExternalWritable := 'False'} : Bool;   // bit opóźnienia reakcji
      bit_hist_close_Z12 { ExternalAccessible := 'False'; ExternalVisible := 'False'; ExternalWritable := 'False'} : Bool;   // bit opóźnienia reakcji
   END_VAR


BEGIN
	(*
	//=============================================================================
	//(JZWiK S.A Radosław Tecmer)
	//(c)Copyright (2021) All Rights Reserved
	//-----------------------------------------------------------------------------
	//Testowane z:   (system docelowy z  FW 4.4)
	//Pakiet inżynierski:   TIA Portal (V14 Sp1 Update 9)
	//Ograniczenia:  ( - )
	//Wymagania:  (minimalne S7-1200 CPU 1215C FW 4.2 .)
	//Funkcjonalnośc: (Sterowanie kierunkiem pompowania Z11 - miasto, 
	                    Z12 - magistrala. W oparciu o sygnał 
	                   wyboru [dbHoldRegSlave_to_MT101.instSygSter_1 - %DB100.DBW52]
	                   0- wyłączone, 1- dosilanie, 2 - przetłaczanie, 3- automat, 
	                   4- ręczne następuje otwarcie właściwej zasuwy. Warunek pracy 
	                   dosilanie zmknięta zasuwa Z10, otwarta Z9. Przetłaczanie warunek
	                   otwarta Z9)
	//-----------------------------------------------------------------------------
	//Zmainy wprowadzone:
	//Wersja  Data       Osoba wprowadzająca zmiany - ekspert
	//01.00.00 17.11.2021 (Tecmer Radosław - twórca) Pieresza wersja 01.00.00
	//=============================================================================
	*)
	
	
	
	
	
	
	
	// Z11 PRZETŁACZANIE
	
	REGION Przetłaczanie
	  // OTWIERANIE
	  // Warunek wystawienia rozkazu na otwarcie Z11
	  IF "dbtags_Sterowanie"."Paramaetry _Zbiorniki".set_strategia_sterowania = 2
	    AND "dbtags_Sterowanie"."Paramaetry _Zbiorniki".set_położenie_Z10 < 2
	    AND "inputZamkniętaZ12"
	    AND "bitH_REM_Z11"
	    AND "bitH_Aut_Man_Z11"
	    AND "inputOtwartaZ11" = FALSE
	    AND %DB10.DBX316.1 // otwarta Z9
	    AND %DB10.DBX316.0 = FALSE // brak awaii Z9
	    AND %DB10.DBX316.7 // tryb automat Z9
	    AND #bit_alarm_magistrala_min = FALSE
	  THEN
	  // 
	    #bit_hist_open_Z11 := TRUE;
	  ELSE
	    #bit_hist_open_Z11 := FALSE;
	  ;
	END_IF;
	
	 "IEC_Timer_OpenZ11_strategia_DB".TON(IN:=#bit_hist_open_Z11,
	                                     PT:=T#10S,
	                                     Q=>#bit_set_open_Z11);
	
	IF #bit_set_open_Z11 THEN
	  // start otwieranie
	  #CMD_Open_Z11 := TRUE;
	ELSE
	  #CMD_Open_Z11 := FALSE;
	  ;
	END_IF;
	
	// ZAMYKANIE
	// Warune na zamykanie Z11
	IF (%DB10.DBX316.1 = FALSE // brak otwarcia Z9
	  OR #bit_alarm_magistrala_min) OR // awaria niskie ciśnienie na magistrali
	  "dbtags_Sterowanie"."Paramaetry _Zbiorniki".set_strategia_sterowania = 1 OR
	  "dbtags_Sterowanie"."Paramaetry _Zbiorniki".set_strategia_sterowania = 0
	  AND "bitH_REM_Z11"
	  AND "bitH_Aut_Man_Z11"
	  AND "inputOtwartaZ11"
	
	THEN 
	  // start zamykanie
	  #bit_hist_close_Z11:= TRUE;
	ELSE
	  #bit_hist_close_Z11 := FALSE;
	  ;
	END_IF;
	
	 "IEC_Timer_Zmykanie Z11_DB".TON(IN:=#bit_hist_close_Z11,
	                                PT:=T#10S,
	                                Q=>#bit_set_close_Z11);
	
	IF #bit_hist_close_Z11 THEN
	  // start na zamykanie
	  #CMD_Close_Z11 := TRUE;
	ELSE
	  #CMD_Close_Z11 := FALSE;
	  ;
	END_IF;
	
	
	
	END_REGION
	
	
	
	
END_FUNCTION_BLOCK

FUNCTION_BLOCK "Strategia sterowaia Z12"
TITLE = Strategia sterowania 
{ S7_Optimized_Access := 'TRUE' }
AUTHOR : rtecmer
VERSION : 0.1
//Funkcja sterowania przełączaniem kieunku pompowania Z11 - przetłaczania kierunek miasto, Z12 - dosilanie w kierunku magistrali
   VAR_INPUT 
      bit_alarm_magistrala_min { ExternalAccessible := 'False'; ExternalVisible := 'False'; ExternalWritable := 'False'} : Bool := false;   // bit alarmmagistrala awaria niskie ciśnienie
   END_VAR

   VAR_IN_OUT 
      CMD_Open_Z12 : Bool;   // znacznik sterowania zamykaniem
      CMD_Close_Z12 : Bool := false;   // znacznik sterowania zamykaniem
   END_VAR

   VAR 
      bit_set_open_Z11 { ExternalAccessible := 'False'; ExternalVisible := 'False'; ExternalWritable := 'False'} : Bool;   // bit inicjacji otwierania zasuwy w trybie strategii
      bit_set_open_Z12 { ExternalAccessible := 'False'; ExternalVisible := 'False'; ExternalWritable := 'False'} : Bool;   // bit inicjacji otwierania zasuwy w trybie strategii
      bit_hist_open_Z11 { ExternalAccessible := 'False'; ExternalVisible := 'False'; ExternalWritable := 'False'} : Bool;   // bit opóźnienia reakcji
      bit_hist_open_Z12 { ExternalAccessible := 'False'; ExternalVisible := 'False'; ExternalWritable := 'False'} : Bool;   // bit opóźnienia reakcji
      bit_set_close_Z11 { ExternalAccessible := 'False'; ExternalVisible := 'False'; ExternalWritable := 'False'} : Bool;   // bit inicjacji otwierania zasuwy w trybie strategii
      bit_set_close_Z12 { ExternalAccessible := 'False'; ExternalVisible := 'False'; ExternalWritable := 'False'} : Bool;   // bit inicjacji otwierania zasuwy w trybie strategii
      bit_hist_close_Z11 { ExternalAccessible := 'False'; ExternalVisible := 'False'; ExternalWritable := 'False'} : Bool;   // bit opóźnienia reakcji
      bit_hist_close_Z12 { ExternalAccessible := 'False'; ExternalVisible := 'False'; ExternalWritable := 'False'} : Bool;   // bit opóźnienia reakcji
   END_VAR


BEGIN
	(*
	//=============================================================================
	//(JZWiK S.A Radosław Tecmer)
	//(c)Copyright (2021) All Rights Reserved
	//-----------------------------------------------------------------------------
	//Testowane z:   (system docelowy z  FW 4.4)
	//Pakiet inżynierski:   TIA Portal (V14 Sp1 Update 9)
	//Ograniczenia:  ( - )
	//Wymagania:  (minimalne S7-1200 CPU 1215C FW 4.2 .)
	//Funkcjonalnośc: (Sterowanie kierunkiem pompowania Z11 - miasto, 
	                    Z12 - magistrala. W oparciu o sygnał 
	                   wyboru [dbHoldRegSlave_to_MT101.instSygSter_1 - %DB100.DBW52]
	                   0- wyłączone, 1- dosilanie, 2 - przetłaczanie, 3- automat, 
	                   4- ręczne następuje otwarcie właściwej zasuwy. Warunek pracy 
	                   dosilanie zmknięta zasuwa Z10, otwarta Z9. Przetłaczanie warunek
	                   otwarta Z9)
	//-----------------------------------------------------------------------------
	//Zmainy wprowadzone:
	//Wersja  Data       Osoba wprowadzająca zmiany - ekspert
	//01.00.00 17.11.2021 (Tecmer Radosław - twórca) Pieresza wersja 01.00.00
	//=============================================================================
	*)
	
	
	
	
	
	// Z12 DOSILANIE 
	
	REGION Dosilanie
	  // OTWIERANIE
	  // Warunek wystawienia rozkazu na otwarcie Z12
	  IF "dbtags_Sterowanie"."Paramaetry _Zbiorniki".set_strategia_sterowania = 1
	    AND "dbtags_Sterowanie"."Paramaetry _Zbiorniki".set_położenie_Z10 < 2
	    AND "inputZamkniętaZ11"
	    AND "bitH_REM_Z12"
	    AND "bitH_Aut_Man_Z12"
	    AND "inputOtwartaZ12" = FALSE
	    AND %DB10.DBX316.1 // otwarta Z9
	    AND %DB10.DBX316.0 = FALSE // brak awarii Z9  
	    AND %DB10.DBX316.7 // tryb automat Z9
	  THEN
	    // 
	    #bit_hist_open_Z12 := TRUE;
	  ELSE
	    #bit_hist_open_Z12 := FALSE;
	    ;
	  END_IF;
	   "IEC_Timer_OpenZ12_DB".TON(IN:=#bit_hist_open_Z12,
	                             PT:=T#10S,
	                             Q=>#bit_set_open_Z12);
	  
	  
	  IF #bit_set_open_Z12  THEN
	    // start otwieranie
	    #CMD_Open_Z12 := TRUE;
	  ELSE
	    #CMD_Open_Z12 := FALSE;
	    ;
	  END_IF;
	  
	  // ZAMYKANIE
	  // Warune na zamykanie Z12
	  IF %DB10.DBX316.1 = FALSE OR  // brak otwarcia Z9
	    "dbtags_Sterowanie"."Paramaetry _Zbiorniki".set_strategia_sterowania = 2 OR
	    "dbtags_Sterowanie"."Paramaetry _Zbiorniki".set_strategia_sterowania = 0
	    AND "bitH_REM_Z12"
	    AND "bitH_Aut_Man_Z12"
	    AND "inputOtwartaZ12"
	
	  THEN
	    // start zamykanie
	    #bit_hist_close_Z12 := TRUE;
	  ELSE
	    #bit_hist_close_Z12 := FALSE;
	    ;
	  END_IF;
	  
	  "IEC_Timer_ZamykanieZ12_DB".TON(IN:=#bit_hist_close_Z12,
	                                  PT:=T#10S,
	                                  Q=>#bit_set_close_Z12);
	  
	  
	  IF #bit_hist_close_Z12 THEN
	    // start na zamykanie
	    #CMD_Close_Z12 := TRUE;
	  ELSE
	    #CMD_Close_Z12 := FALSE;
	    ;
	  END_IF;
	  
	  
	  
	END_REGION
	
END_FUNCTION_BLOCK

FUNCTION_BLOCK "Alarm-Pompownia-Sucho-Max"
TITLE = reakcja na niskie ciśnienie na ssaniu
{ S7_Optimized_Access := 'TRUE' }
AUTHOR : rtecmer
VERSION : 0.1
//Funkcja realizuje zatrzymanie pomp z powodu niskiego ciśnienia ssania
   VAR_OUTPUT 
      bit_on_alarm_bar_max_pompownia { ExternalWritable := 'False'} : Bool;   // bit alarmu maksymalnego ciśnienia na pompowni
   END_VAR

   VAR 
      bit_max_pompownia { ExternalAccessible := 'False'; ExternalVisible := 'False'; ExternalWritable := 'False'} : Bool := false;   // bit detekcji wysokiego ciśnienia pompownia B7
      bit_normalne_pompownia { ExternalAccessible := 'False'; ExternalVisible := 'False'; ExternalWritable := 'False'} : Bool := false;   // bit detekcji normalnego cisnienia pompownia
      "bit_max _bar_B7" { ExternalAccessible := 'False'; ExternalVisible := 'False'; ExternalWritable := 'False'} : Bool := false;   // bit zaistnienia max ciśnienia pompownia B7
      bit_off_alarm_max_pompownia { ExternalAccessible := 'False'; ExternalVisible := 'False'; ExternalWritable := 'False'} : Bool;   // koniec alarmu max B7 pompownia
   END_VAR


BEGIN
	(*
	//=============================================================================
	//(JZWiK S.A Radosław Tecmer)
	//(c)Copyright (2021) All Rights Reserved
	//-----------------------------------------------------------------------------
	//Testowane z:   (system docelowy z  FW 4.4)
	//Pakiet inżynierski:   TIA Portal (V14 Sp1 Update 9)
	//Ograniczenia:  ( - )
	//Wymagania:  (minimalne S7-1200 CPU 1215C FW 4.2 .)
	//Funkcjonalnośc: (Kontrola ciśnienia max przepompownia 
	                   Ustawienie i kasowanie bitu awarii od max ciśnienia
	                   na pompowni.)
	//-----------------------------------------------------------------------------
	//Zmainy wprowadzone:
	//Wersja  Data       Osoba wprowadzająca zmiany - ekspert
	//01.00.00 17.11.2021 (Tecmer Radosław - twórca) Pieresza wersja 01.00.00
	//=============================================================================
	*)
	
	
	
	
	
	
	
	
	REGION Kontrola ciśnienia pompownia - ciśnienie max
	  // Kontrola max pompownia ustawione alarmowe 9.0
	  IF "dbdane".act_Value_B7 >= "db10organizacyjna".set_press_bar_Max THEN
	    // Ustaw bit alarmowe ciśnienie na B7
	    #"bit_max _bar_B7" := TRUE;
	    #bit_normalne_pompownia := FALSE;
	  ELSE
	    #bit_normalne_pompownia := TRUE;
	    ;
	  END_IF;
	  
	  
	  //warunek koniec alarmu max
	  IF "dbdane".act_Value_B7 <= ("db10organizacyjna".set_press_bar_Max - 0.2) THEN
	    // ustaw bit ciśnienie poprawne
	    #bit_normalne_pompownia := TRUE;
	    ;
	  END_IF;
	  
	  // kasowania alarmu
	  IF #bit_off_alarm_max_pompownia THEN
	    // kasowanie alarmu ssania
	    #bit_on_alarm_bar_max_pompownia := FALSE;
	    #"bit_max _bar_B7" := FALSE;
	    
	  END_IF;
	  
	  // Histerez ana ustawienie alarmu max bar
	  "IEC_Timer_B7max_bar_DB".TON(IN:=#"bit_max _bar_B7",
	                               PT:=T#10S,
	                               Q=>#bit_on_alarm_bar_max_pompownia);
	  
	 "IEC_Timer_B7max_off_alarm_DB".TON(IN:=#bit_normalne_pompownia,
	                                   PT:=T#10S,
	                                   Q=>#bit_off_alarm_max_pompownia);
	
	
	  
	  
	  
	  
	END_REGION
	
	
END_FUNCTION_BLOCK

FUNCTION_BLOCK "Strategia sterowania Pompownia"   // FB4, LAD
TITLE = Wygór metody sterowania
{ S7_Optimized_Access := 'TRUE' }
AUTHOR : rtecmer
VERSION : 0.1
// Wybór strategi "Dosilanie" - Kierunek pompowania na magistralę poprzez Z12, "Przetłaczanie" - Kierunek na miasto przez Z11,  "Automat" - sterownik PLC decyduje o kierunku toczenia, "Ręczne" -  Manualie sterowanie przez operatora. Sterowanie zależne od położenia Z9 (Szafa PLC Zasuwy)
// stored: AutoNumber true, IsIECCheckEnabled false, IsRetainMemResEnabled false, MemoryReserve 100, SetENOAutomatically false, UDAEnableTagReadback false
   VAR_INPUT
      tempStrategia_Pompownia : Int;   // Słowo strategii przechwyconej w FB24
      "bit_alarm_magistrala _min" : Bool;   // bit alarmu niskie ciśniei na magistrali
      bit_off_alarm_magistrala_niskie : Bool;   // bit wyłaczenia alarmu magistrali niskie
   END_VAR
   VAR_IN_OUT
      "Strategia Pompownia" : Int;
   END_VAR
   VAR
      tmp_on_alarm { ExternalAccessible := 'False'; ExternalVisible := 'False'; ExternalWritable := 'False'} : Bool;
      tmp_off_alarm { ExternalAccessible := 'False'; ExternalVisible := 'False'; ExternalWritable := 'False'} : Bool;
      memTriger_set_Strategia { ExternalAccessible := 'False'; ExternalVisible := 'False'; ExternalWritable := 'False'} : Bool;
      memTriger_reset_Strategia { ExternalAccessible := 'False'; ExternalVisible := 'False'; ExternalWritable := 'False'} : Bool;
      test { ExternalAccessible := 'False'; ExternalVisible := 'False'; ExternalWritable := 'False'} : Bool;
   END_VAR
   VAR CONSTANT
      "strategia awaria" : Int := 1;
   END_VAR
   VAR_TEMP   // added for the SCL form of the ladder/FBD networks
      _w1 : Bool;
      _w2 : Bool;
   END_VAR
BEGIN

REGION Network 1: Koniec awarii magistrali
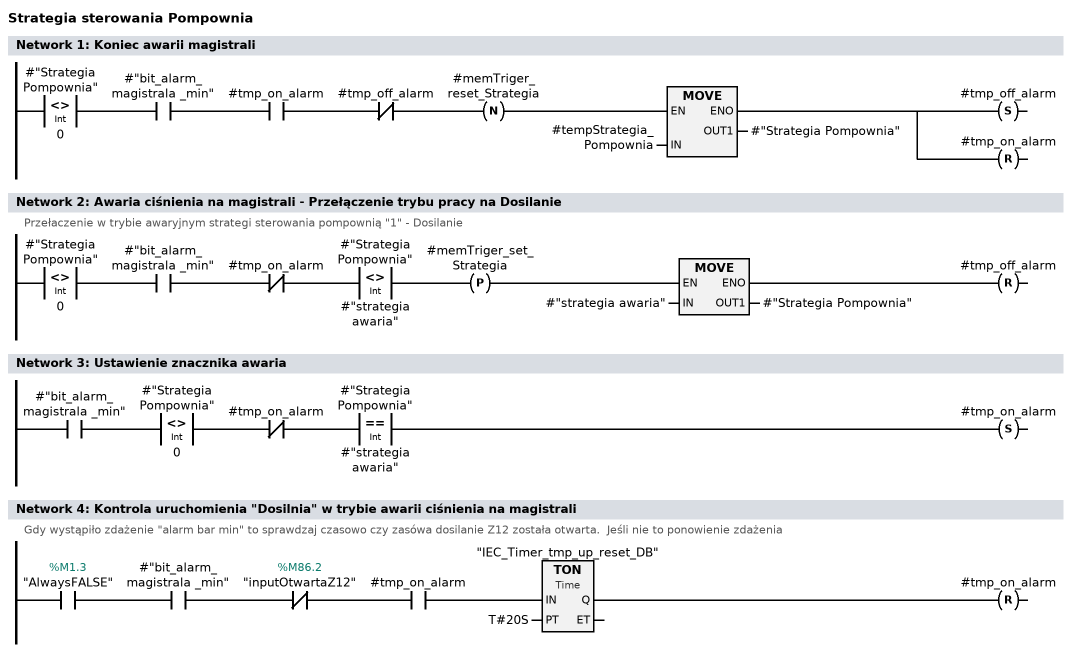
   RUNG wire#powerrail
      { S7_Templates := "SrcType := Int" } NE_Contact(in1 := #"Strategia Pompownia", in2 := 0)
      Contact( #"bit_alarm_magistrala _min" )
      Contact( #tmp_on_alarm )
      I_Contact( #tmp_off_alarm )
      N_Trig( #memTriger_reset_Strategia )
      Move(in := #tempStrategia_Pompownia, out1 => #"Strategia Pompownia")
      wire#w1
      S_Coil( #tmp_off_alarm )
   END_RUNG
   RUNG wire#w1
      R_Coil( #tmp_on_alarm )
   END_RUNG
   // the same network as SCL:
   #_w1 := (#"Strategia Pompownia" <> 0) AND #"bit_alarm_magistrala _min" AND #tmp_on_alarm AND NOT #tmp_off_alarm;
   #_w2 := NOT #_w1 AND #memTriger_reset_Strategia;   // falling edge
   #memTriger_reset_Strategia := #_w1;
   IF #_w2 THEN
       #"Strategia Pompownia" := #tempStrategia_Pompownia;
       #tmp_off_alarm := TRUE;
       #tmp_on_alarm := FALSE;
   END_IF;
END_REGION

REGION Network 2: Awaria ciśnienia na magistrali - Przełączenie trybu pracy na Dosilanie
   // Przełaczenie w trybie awaryjnym strategi sterowania pompownią "1" - Dosilanie
   RUNG wire#powerrail
      { S7_Templates := "SrcType := Int" } NE_Contact(in1 := #"Strategia Pompownia", in2 := 0)
      Contact( #"bit_alarm_magistrala _min" )
      I_Contact( #tmp_on_alarm )
      { S7_Templates := "SrcType := Int" } NE_Contact(in1 := #"Strategia Pompownia", in2 := #"strategia awaria")
      P_Trig( #memTriger_set_Strategia )
      Move(in := #"strategia awaria", out1 => #"Strategia Pompownia")
      R_Coil( #tmp_off_alarm )
   END_RUNG
   // the same network as SCL:
   #_w1 := (#"Strategia Pompownia" <> 0) AND #"bit_alarm_magistrala _min" AND NOT #tmp_on_alarm AND (#"Strategia Pompownia" <> #"strategia awaria");
   #_w2 := #_w1 AND NOT #memTriger_set_Strategia;   // rising edge
   #memTriger_set_Strategia := #_w1;
   IF #_w2 THEN
       #"Strategia Pompownia" := #"strategia awaria";
       #tmp_off_alarm := FALSE;
   END_IF;
END_REGION

REGION Network 3: Ustawienie znacznika awaria
   RUNG wire#powerrail
      Contact( #"bit_alarm_magistrala _min" )
      { S7_Templates := "SrcType := Int" } NE_Contact(in1 := #"Strategia Pompownia", in2 := 0)
      I_Contact( #tmp_on_alarm )
      { S7_Templates := "SrcType := Int" } EQ_Contact(in1 := #"Strategia Pompownia", in2 := #"strategia awaria")
      S_Coil( #tmp_on_alarm )
   END_RUNG
   // the same network as SCL:
   IF #"bit_alarm_magistrala _min" AND (#"Strategia Pompownia" <> 0) AND NOT #tmp_on_alarm AND (#"Strategia Pompownia" = #"strategia awaria") THEN
       #tmp_on_alarm := TRUE;
   END_IF;
END_REGION

REGION Network 4: Kontrola uruchomienia "Dosilnia" w trybie awarii ciśnienia na magistrali
   // Gdy wystąpiło zdażenie "alarm bar min" to sprawdzaj czasowo czy zasówa dosilanie Z12 została otwarta.  Jeśli nie to ponowienie zdażenia
   RUNG wire#powerrail
      Contact( "AlwaysFALSE" )
      Contact( #"bit_alarm_magistrala _min" )
      I_Contact( "inputOtwartaZ12" )
      Contact( #tmp_on_alarm )
      { S7_Templates := "time_type := Time" } "IEC_Timer_tmp_up_reset_DB".TON(pt := T#20S, et =>)
      R_Coil( #tmp_on_alarm )
   END_RUNG
   // the same network as SCL:
   "IEC_Timer_tmp_up_reset_DB".TON(IN := "AlwaysFALSE" AND #"bit_alarm_magistrala _min" AND NOT "inputOtwartaZ12" AND #tmp_on_alarm,
                           PT := T#20S);
   IF "IEC_Timer_tmp_up_reset_DB".Q THEN #tmp_on_alarm := FALSE; END_IF;
END_REGION
END_FUNCTION_BLOCK

FUNCTION "Sterowniki_Z11_Z12" : Void   // FC30, LAD
TITLE = Driver napedów zasuw Z11, Z12
{ S7_Optimized_Access := 'TRUE' }
AUTHOR : rtecmer
VERSION : 0.1
// Funkcje sterujące napędami w trybie zdalnym, lokalnym
// stored: AutoNumber true, IsIECCheckEnabled false, SetENOAutomatically false, UDAEnableTagReadback false
BEGIN

REGION Network 1: Zasuwa Z11
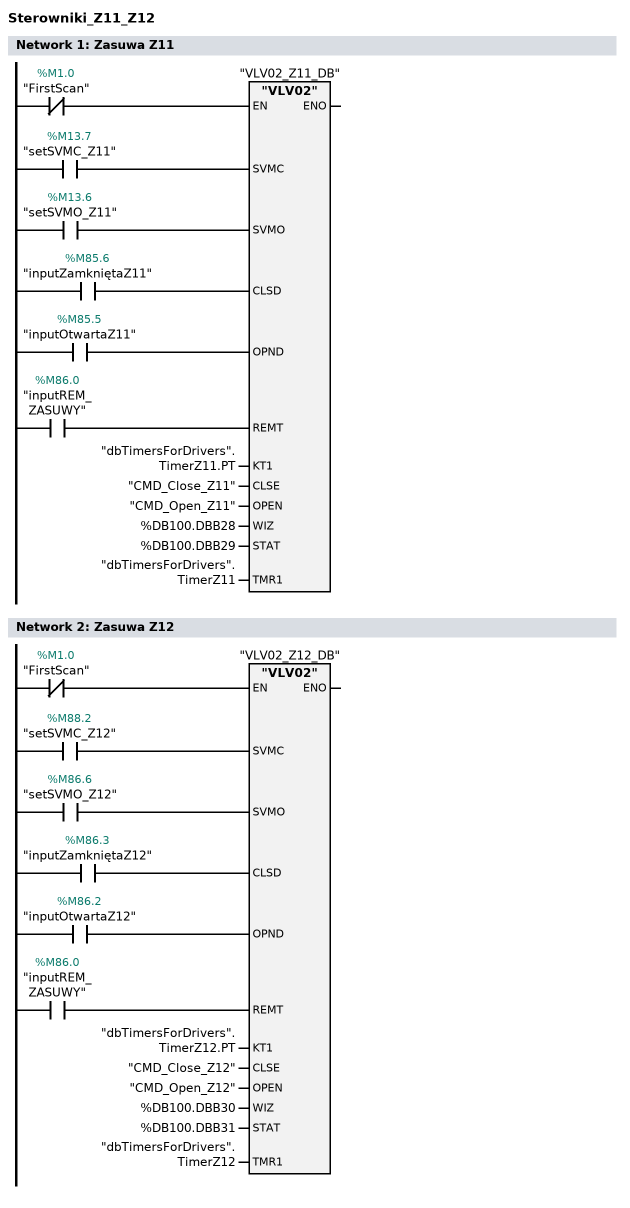
   RUNG wire#powerrail
      I_Contact( "FirstScan" )
      "VLV02_Z11_DB"(SVMC := wire#w1, SVMO := wire#w2, CLSD := wire#w3, OPND := wire#w4, REMT := wire#w5, KT1 := "dbTimersForDrivers".TimerZ11.PT, CLSE := "CMD_Close_Z11", OPEN := "CMD_Open_Z11", WIZ := %DB100.DBB28, STAT := %DB100.DBB29, TMR1 := "dbTimersForDrivers".TimerZ11)
   END_RUNG
   RUNG wire#powerrail
      Contact( "setSVMC_Z11" )
   END_RUNG wire#w1
   RUNG wire#powerrail
      Contact( "setSVMO_Z11" )
   END_RUNG wire#w2
   RUNG wire#powerrail
      Contact( "inputZamkniętaZ11" )
   END_RUNG wire#w3
   RUNG wire#powerrail
      Contact( "inputOtwartaZ11" )
   END_RUNG wire#w4
   RUNG wire#powerrail
      Contact( "inputREM_ZASUWY" )
   END_RUNG wire#w5
   // the same network as SCL:
   IF NOT "FirstScan" THEN
       "VLV02_Z11_DB"(SVMC := "setSVMC_Z11",   // "VLV02"
                      SVMO := "setSVMO_Z11",
                      CLSD := "inputZamkniętaZ11",
                      OPND := "inputOtwartaZ11",
                      REMT := "inputREM_ZASUWY",
                      KT1 := "dbTimersForDrivers".TimerZ11.PT,
                      CLSE := "CMD_Close_Z11",
                      OPEN := "CMD_Open_Z11",
                      WIZ := %DB100.DBB28,
                      STAT := %DB100.DBB29,
                      TMR1 := "dbTimersForDrivers".TimerZ11);
   END_IF;
END_REGION

REGION Network 2: Zasuwa Z12
   RUNG wire#powerrail
      I_Contact( "FirstScan" )
      "VLV02_Z12_DB"(SVMC := wire#w1, SVMO := wire#w2, CLSD := wire#w3, OPND := wire#w4, REMT := wire#w5, KT1 := "dbTimersForDrivers".TimerZ12.PT, CLSE := "CMD_Close_Z12", OPEN := "CMD_Open_Z12", WIZ := %DB100.DBB30, STAT := %DB100.DBB31, TMR1 := "dbTimersForDrivers".TimerZ12)
   END_RUNG
   RUNG wire#powerrail
      Contact( "setSVMC_Z12" )
   END_RUNG wire#w1
   RUNG wire#powerrail
      Contact( "setSVMO_Z12" )
   END_RUNG wire#w2
   RUNG wire#powerrail
      Contact( "inputZamkniętaZ12" )
   END_RUNG wire#w3
   RUNG wire#powerrail
      Contact( "inputOtwartaZ12" )
   END_RUNG wire#w4
   RUNG wire#powerrail
      Contact( "inputREM_ZASUWY" )
   END_RUNG wire#w5
   // the same network as SCL:
   IF NOT "FirstScan" THEN
       "VLV02_Z12_DB"(SVMC := "setSVMC_Z12",   // "VLV02"
                      SVMO := "setSVMO_Z12",
                      CLSD := "inputZamkniętaZ12",
                      OPND := "inputOtwartaZ12",
                      REMT := "inputREM_ZASUWY",
                      KT1 := "dbTimersForDrivers".TimerZ12.PT,
                      CLSE := "CMD_Close_Z12",
                      OPEN := "CMD_Open_Z12",
                      WIZ := %DB100.DBB30,
                      STAT := %DB100.DBB31,
                      TMR1 := "dbTimersForDrivers".TimerZ12);
   END_IF;
END_REGION
END_FUNCTION

FUNCTION_BLOCK "VLV02"   // FB5, LAD
TITLE = Valve driver 02
{ S7_Optimized_Access := 'FALSE' }
AUTHOR : RTecmer
VERSION : 0.2
// Driver for two-position drives
// Slowo STATUSU Napedu
// STAT - Prawy Byte
// WIZ  - Lewy Byte
//  
//   -STAT wektor stanu zaworu
//     -bit 0- alarm                                  (sygnal do SCADA)
//     -bit 1- zawor otwarty                    (sygnal do SCADA)
//     -bit 2-sterowanie zdal=1 loc=0 (sygnal do SCADA)
//     -bit 3- zawor zamkniety               (sygnal do SCADA)
//     -bit 4-otwieranie reczne              (sygnal z SCADA)
//     -bit 5-zamykanie reczne              (sygnal z SCADA)
//     -bit 6-alarm reset                        (sygnal z SCADA
//     -bit 8-auto= 1man=0                  (sygnal z SCADA)
//   -SUPV 
//   -CLSD zawor zamkniety                    - wejscie
//   -OPND zawor otwarty                        - wejscie
//   -REMT sterowanie zdal=1 loc=0      - wejscie
//   -OPEN otwarcie                                  - wyjscie
//   -CLSE zamkniecie                              - wyjscie
//   - TIM1 czas otwierania  
//   - TIM2 czas zamykania
// stored: AutoNumber true, IsIECCheckEnabled false, SetENOAutomatically false, UDAEnableTagReadback false
   VAR_INPUT
      SVMC : Bool;   // Automat na zamykanie
      SVMO { ExternalVisible := 'False'} : Bool;   // Automat na otwieranie
      CLSD : Bool;   // Zamknięta
      OPND : Bool;   // Otwarta
      REMT : Bool;   // Sterowanie zdalne =1, remontowe=0
      KT1 : Time;   // Czas timera
   END_VAR
   VAR_IN_OUT
      CLSE { ExternalAccessible := 'False'; ExternalVisible := 'False'; ExternalWritable := 'False'} : Bool;   // Wyjście zamykanie
      OPEN { ExternalAccessible := 'False'; ExternalVisible := 'False'; ExternalWritable := 'False'} : Bool;   // Wyjście Otwieranie
      WIZ : Byte;   // Wektor SCADA
      STAT : Byte;   // Wektor statusu napędu
      TMR1 : TON_TIME;
   END_VAR
BEGIN

REGION Network 1
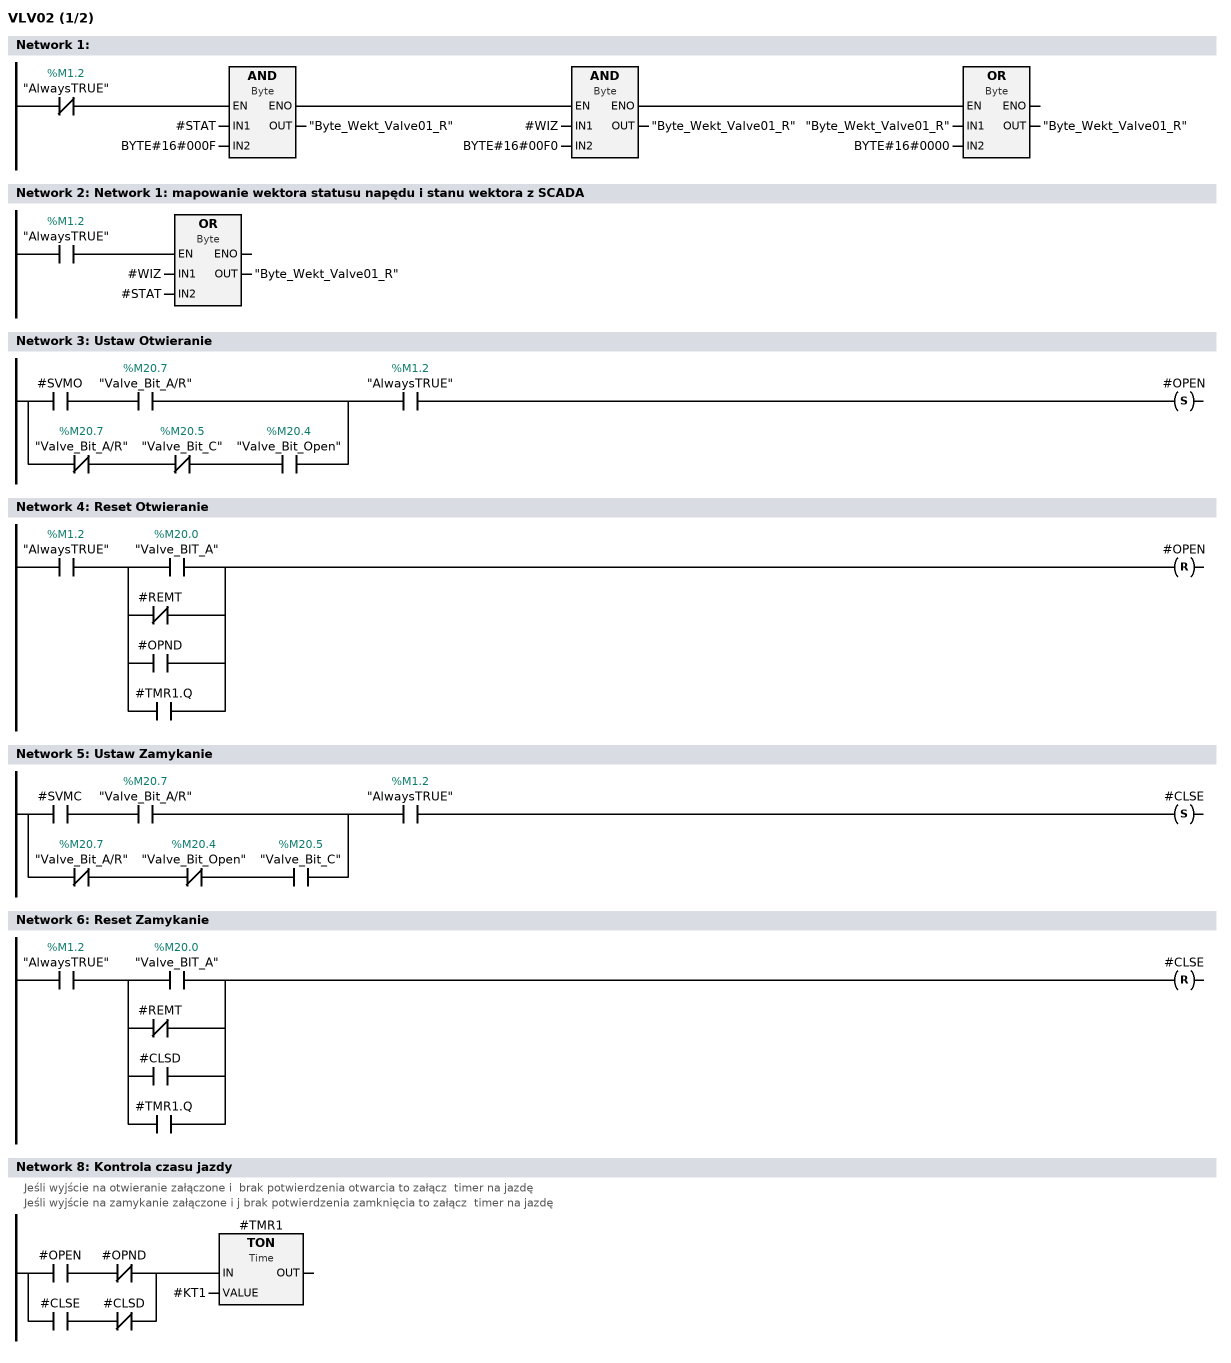
   IF NOT "AlwaysTRUE" THEN
       "Byte_Wekt_Valve01_R" := #STAT AND BYTE#16#000F;
       "Byte_Wekt_Valve01_R" := #WIZ AND BYTE#16#00F0;
       "Byte_Wekt_Valve01_R" := "Byte_Wekt_Valve01_R" OR BYTE#16#0000;
   END_IF;
END_REGION

REGION Network 2: Network 1: mapowanie wektora statusu napędu i stanu wektora z SCADA
   IF "AlwaysTRUE" THEN "Byte_Wekt_Valve01_R" := #WIZ OR #STAT; END_IF;
END_REGION

REGION Network 3: Ustaw Otwieranie
   RUNG wire#powerrail
      Contact( #SVMO )
      Contact( "Valve_Bit_A/R" )
      wire#w1
      Contact( "AlwaysTRUE" )
      S_Coil( #OPEN )
   END_RUNG
   RUNG wire#powerrail
      I_Contact( "Valve_Bit_A/R" )
      I_Contact( "Valve_Bit_C" )
      Contact( "Valve_Bit_Open" )
   END_RUNG wire#w1
   // the same network as SCL:
   IF ((#SVMO AND "Valve_Bit_A/R") OR (NOT "Valve_Bit_A/R" AND NOT "Valve_Bit_C" AND "Valve_Bit_Open")) AND "AlwaysTRUE" THEN
       #OPEN := TRUE;
   END_IF;
END_REGION

REGION Network 4: Reset Otwieranie
   RUNG wire#powerrail
      Contact( "AlwaysTRUE" )
      wire#w1
      Contact( "Valve_BIT_A" )
      wire#w2
      R_Coil( #OPEN )
   END_RUNG
   RUNG wire#w1
      I_Contact( #REMT )
   END_RUNG wire#w2
   RUNG wire#w1
      Contact( #OPND )
   END_RUNG wire#w2
   RUNG wire#w1
      Contact( #TMR1.Q )
   END_RUNG wire#w2
   // the same network as SCL:
   IF "AlwaysTRUE" AND ("Valve_BIT_A" OR NOT #REMT OR #OPND OR #TMR1.Q) THEN #OPEN := FALSE; END_IF;
END_REGION

REGION Network 5: Ustaw Zamykanie
   RUNG wire#powerrail
      Contact( #SVMC )
      Contact( "Valve_Bit_A/R" )
      wire#w1
      Contact( "AlwaysTRUE" )
      S_Coil( #CLSE )
   END_RUNG
   RUNG wire#powerrail
      I_Contact( "Valve_Bit_A/R" )
      I_Contact( "Valve_Bit_Open" )
      Contact( "Valve_Bit_C" )
   END_RUNG wire#w1
   // the same network as SCL:
   IF ((#SVMC AND "Valve_Bit_A/R") OR (NOT "Valve_Bit_A/R" AND NOT "Valve_Bit_Open" AND "Valve_Bit_C")) AND "AlwaysTRUE" THEN
       #CLSE := TRUE;
   END_IF;
END_REGION

REGION Network 6: Reset Zamykanie
   RUNG wire#powerrail
      Contact( "AlwaysTRUE" )
      wire#w1
      Contact( "Valve_BIT_A" )
      wire#w2
      R_Coil( #CLSE )
   END_RUNG
   RUNG wire#w1
      I_Contact( #REMT )
   END_RUNG wire#w2
   RUNG wire#w1
      Contact( #CLSD )
   END_RUNG wire#w2
   RUNG wire#w1
      Contact( #TMR1.Q )
   END_RUNG wire#w2
   // the same network as SCL:
   IF "AlwaysTRUE" AND ("Valve_BIT_A" OR NOT #REMT OR #CLSD OR #TMR1.Q) THEN #CLSE := FALSE; END_IF;
END_REGION

REGION Network 8: Kontrola czasu jazdy
   // Jeśli wyjście na otwieranie załączone i  brak potwierdzenia otwarcia to załącz  timer na jazdę
   // Jeśli wyjście na zamykanie załączone i j brak potwierdzenia zamknięcia to załącz  timer na jazdę
   #TMR1(IN := (#OPEN AND NOT #OPND) OR (#CLSE AND NOT #CLSD), PT := #KT1);   // TON coil
END_REGION

REGION Network 9: Bit alarm ustaw
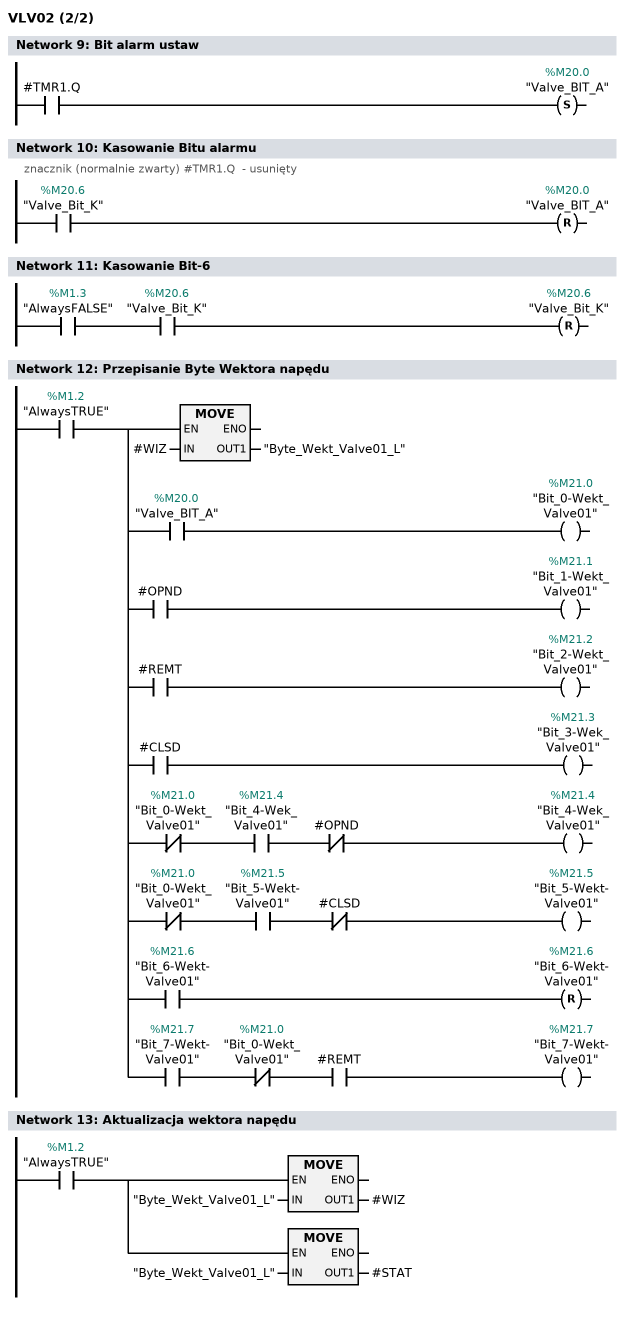
   RUNG wire#powerrail
      Contact( #TMR1.Q )
      S_Coil( "Valve_BIT_A" )
   END_RUNG
   // the same network as SCL:
   IF #TMR1.Q THEN "Valve_BIT_A" := TRUE; END_IF;
END_REGION

REGION Network 10: Kasowanie Bitu alarmu
   // znacznik (normalnie zwarty) #TMR1.Q  - usunięty
   RUNG wire#powerrail
      Contact( "Valve_Bit_K" )
      R_Coil( "Valve_BIT_A" )
   END_RUNG
   // the same network as SCL:
   IF "Valve_Bit_K" THEN "Valve_BIT_A" := FALSE; END_IF;
END_REGION

REGION Network 11: Kasowanie Bit-6
   RUNG wire#powerrail
      Contact( "AlwaysFALSE" )
      Contact( "Valve_Bit_K" )
      R_Coil( "Valve_Bit_K" )
   END_RUNG
   // the same network as SCL:
   IF "AlwaysFALSE" AND "Valve_Bit_K" THEN "Valve_Bit_K" := FALSE; END_IF;
END_REGION

REGION Network 12: Przepisanie Byte Wektora napędu
   RUNG wire#powerrail
      Contact( "AlwaysTRUE" )
      wire#w1
      { S7_GenerateENO := "TRUE" } Move(in := #WIZ, out1 => "Byte_Wekt_Valve01_L")
   END_RUNG
   RUNG wire#w1
      Contact( "Valve_BIT_A" )
      Coil( "Bit_0-Wekt_Valve01" )
   END_RUNG
   RUNG wire#w1
      Contact( #OPND )
      Coil( "Bit_1-Wekt_Valve01" )
   END_RUNG
   RUNG wire#w1
      Contact( #REMT )
      Coil( "Bit_2-Wekt_Valve01" )
   END_RUNG
   RUNG wire#w1
      Contact( #CLSD )
      Coil( "Bit_3-Wek_Valve01" )
   END_RUNG
   RUNG wire#w1
      I_Contact( "Bit_0-Wekt_Valve01" )
      Contact( "Bit_4-Wek_Valve01" )
      I_Contact( #OPND )
      Coil( "Bit_4-Wek_Valve01" )
   END_RUNG
   RUNG wire#w1
      I_Contact( "Bit_0-Wekt_Valve01" )
      Contact( "Bit_5-Wekt-Valve01" )
      I_Contact( #CLSD )
      Coil( "Bit_5-Wekt-Valve01" )
   END_RUNG
   RUNG wire#w1
      Contact( "Bit_6-Wekt-Valve01" )
      R_Coil( "Bit_6-Wekt-Valve01" )
   END_RUNG
   RUNG wire#w1
      Contact( "Bit_7-Wekt-Valve01" )
      I_Contact( "Bit_0-Wekt_Valve01" )
      Contact( #REMT )
      Coil( "Bit_7-Wekt-Valve01" )
   END_RUNG
   // the same network as SCL:
   IF "AlwaysTRUE" THEN "Byte_Wekt_Valve01_L" := #WIZ; END_IF;
   "Bit_0-Wekt_Valve01" := "AlwaysTRUE" AND "Valve_BIT_A";
   "Bit_1-Wekt_Valve01" := "AlwaysTRUE" AND #OPND;
   "Bit_2-Wekt_Valve01" := "AlwaysTRUE" AND #REMT;
   "Bit_3-Wek_Valve01" := "AlwaysTRUE" AND #CLSD;
   "Bit_4-Wek_Valve01" := "AlwaysTRUE" AND NOT "Bit_0-Wekt_Valve01" AND "Bit_4-Wek_Valve01" AND NOT #OPND;
   "Bit_5-Wekt-Valve01" := "AlwaysTRUE" AND NOT "Bit_0-Wekt_Valve01" AND "Bit_5-Wekt-Valve01" AND NOT #CLSD;
   IF "AlwaysTRUE" AND "Bit_6-Wekt-Valve01" THEN "Bit_6-Wekt-Valve01" := FALSE; END_IF;
   "Bit_7-Wekt-Valve01" := "AlwaysTRUE" AND "Bit_7-Wekt-Valve01" AND NOT "Bit_0-Wekt_Valve01" AND #REMT;
END_REGION

REGION Network 13: Aktualizacja wektora napędu
   RUNG wire#powerrail
      Contact( "AlwaysTRUE" )
      wire#w1
      { S7_GenerateENO := "TRUE" } Move(in := "Byte_Wekt_Valve01_L", out1 => #WIZ)
   END_RUNG
   RUNG wire#w1
      { S7_GenerateENO := "TRUE" } Move(in := "Byte_Wekt_Valve01_L", out1 => #STAT)
   END_RUNG
   // the same network as SCL:
   IF "AlwaysTRUE" THEN
       #WIZ := "Byte_Wekt_Valve01_L";
       #STAT := "Byte_Wekt_Valve01_L";
   END_IF;
END_REGION
END_FUNCTION_BLOCK

FUNCTION_BLOCK "Konwertowanie parametrów z falownika ModbusRTU"
{ S7_Optimized_Access := 'TRUE' }
AUTHOR : rtecmer
VERSION : 0.1
   VAR_INPUT 
      received_Inver_setpoint_ref_416020 { ExternalAccessible := 'False'; ExternalVisible := 'False'; ExternalWritable := 'False'} : Int;
      received_Inver_Frequency_416130 { ExternalAccessible := 'False'; ExternalVisible := 'False'; ExternalWritable := 'False'} : Int;
      received_Inver_MotorCurrent_416140 { ExternalAccessible := 'False'; ExternalVisible := 'False'; ExternalWritable := 'False'} : Int;
      received_Inver_NomCurrent_416360 { ExternalAccessible := 'False'; ExternalVisible := 'False'; ExternalWritable := 'False'} : Int;
      received_Inver_MaxCurrent_416370 { ExternalAccessible := 'False'; ExternalVisible := 'False'; ExternalWritable := 'False'} : Int;
      received_Inver_InDigit_416600 { ExternalAccessible := 'False'; ExternalVisible := 'False'; ExternalWritable := 'False'} : Int;
      received_Inver_OverTemp_415040 { ExternalAccessible := 'False'; ExternalVisible := 'False'; ExternalWritable := 'False'} : Int;
      received_Inver_OverVolts_415050 { ExternalAccessible := 'False'; ExternalVisible := 'False'; ExternalWritable := 'False'} : Int;
   END_VAR

   VAR_OUTPUT 
      Setpoint_Inverter { ExternalAccessible := 'False'; ExternalVisible := 'False'; ExternalWritable := 'False'} : Real;   // Wartość zadana Hz odczytane z Modbus
      Frequency_inverter { ExternalAccessible := 'False'; ExternalVisible := 'False'; ExternalWritable := 'False'} : Real;   // Aktualne Hz silniku odczytane z Modbus
      MotorCurrent_Inverter { ExternalAccessible := 'False'; ExternalVisible := 'False'; ExternalWritable := 'False'} : Real;   // Prąd na silniku zasilanym z falownika odczytane z Modbus
      NormalCurrent_Inverter { ExternalAccessible := 'False'; ExternalVisible := 'False'; ExternalWritable := 'False'} : Real;   // Prąd nominalny falownika odczytane z Modbus
      MaxCurrent_Inverter { ExternalAccessible := 'False'; ExternalVisible := 'False'; ExternalWritable := 'False'} : Real;   // Prad Max krótkotrwały odczytane z Modbus
      OverTemp_Inverter { ExternalAccessible := 'False'; ExternalVisible := 'False'; ExternalWritable := 'False'} : Word;
      OverVolta_Inverter { ExternalAccessible := 'False'; ExternalVisible := 'False'; ExternalWritable := 'False'} : Word;
   END_VAR

   VAR_TEMP 
      tmp_1 : Real;
      tmp_2 : Real;
      tmp_3 : Real;
      tmp_4 : Real;
      tmp_5 : Real;
      tmp_6 : Real;
      tmp_7 : Real;
      tmp_8 : Real;
      tmp_9 : Real;
      tmp_10 : Real;
   END_VAR


BEGIN
	(*
	//=============================================================================
	//(JZWiK S.A Radosław Tecmer)
	//(c)Copyright (2021) All Rights Reserved
	//-----------------------------------------------------------------------------
	//Testowane z:   (system docelowy z  FW 4.4)
	//Pakiet inżynierski:   TIA Portal (V14 Sp1 Update 9)
	//Ograniczenia:  ( - )
	//Wymagania:  (minimalne S7-1200 CPU 1215C FW 4.2 .)
	//Funkcjonalnośc: (Konwersja i przeliczenie wartości pobranych  z Modbus RTU 
	//                  na wartości rzeczywiste)
	//-----------------------------------------------------------------------------
	//Zmainy wprowadzone:
	//Wersja  Data       Osoba wprowadzająca zmiany - ekspert
	//01.00.00 11.01.2022 (Tecmer Radosław - twórca) Pieresza wersja 01.00.00
	//=============================================================================
	*)
	
	
	//Wartości indexów zgodnie z dokumentacją Danfoss FC51 Programing Guide:
	//index 2 | mnożnik 10; index 1 | mnożnik 100; index 0 | mnożnik 0
	//index -1 | mnożnik 0.1; index -2 | mnożnik 0.01; index -3 | mnożnik 0.001
	//index -4 | mnożnik 0.0001; index -5 | mnożnik 0.00001
	
	REGION Setpoint Inverter P1-P4
	  // Wyliczanie wartości 
	  #tmp_1 := INT_TO_REAL (#received_Inver_setpoint_ref_416020 );
	  #tmp_2 := (#tmp_1 * 0.1) * 0.01;
	  #Setpoint_Inverter := SCALE_X_REAL(MIN := 0.0,
	                                           VALUE := #tmp_2,
	                                           MAX := 50.0);
	  
	END_REGION
	
	REGION Frequecy Act. Inverter P1-P4
	  // Wyliczanie wartości
	  #tmp_3 := INT_TO_REAL(#received_Inver_Frequency_416130) ;
	  #tmp_4 := (#tmp_3 * 0.1);
	  #Frequency_inverter := #tmp_4;
	  
	END_REGION
	
	REGION Motor Current from Inverter P1-P4
	  // Wyliczanie wartości
	  #tmp_5 := INT_TO_REAL(#received_Inver_MotorCurrent_416140);
	  #tmp_6 := (#tmp_5 * 0.01);
	  #MotorCurrent_Inverter := #tmp_6;
	  
	END_REGION
	
	REGION Nominal Current Inverter P1-P4
	  // Wyliczanie wartości
	  #tmp_7 := INT_TO_REAL(#received_Inver_NomCurrent_416360 );
	  #tmp_8 := (#tmp_7 * 0.01);
	  #NormalCurrent_Inverter := #tmp_8;
	  
	END_REGION
	
	REGION Max Current Inverter P1-P4
	  // Wyliczanie wartości
	  #tmp_9 := INT_TO_REAL(#received_Inver_MaxCurrent_416370 );
	  #tmp_10 := (#tmp_9 * 0.01);
	  #MaxCurrent_Inverter := #tmp_10;
	  
	END_REGION
	
	
	#OverTemp_Inverter:= #received_Inver_OverTemp_415040;
	#OverVolta_Inverter:= #received_Inver_OverVolts_415050;
	
	
END_FUNCTION_BLOCK

FUNCTION_BLOCK "Sterowania bez falownika"   // FB18, LAD
TITLE = Sterowania bez falownika
{ S7_Optimized_Access := 'TRUE' }
AUTHOR : rtecmer
VERSION : 0.1
// Sterowanie awaryjne układemw w wypadku awarii falownika.
// Sterowanie napędami z sieci. 
// Załączenie od sygnału  InputWarning_L_PID. jest to bit ustawiany przez regulator PID  wyliczany na podstawie wartości zadanej tlenu + wartość współczynnika .
// Wyłaczenie natępuje po osiągnięciu "Górnego progu tymczasowego". 
// Praca kompresorów z wyrównaniem liczników pracy.
// Jednocześnie pracuje tylko jeden kompresor.
// Sterowanie awaryjne układemw w wypadku awarii falownika.
// Sterowanie napędami z sieci. 
// Załączenie od sygnału  InputWarning_L_PID. jest to bit ustawiany przez regulator PID  wyliczany na podstawie wartości zadanej bar + wartość współczynnika .
// Wyłaczenie natępuje po osiągnięciu "Górnego progu tymczasowego". 
// Praca kompresorów z wyrównaniem liczników pracy.
// Jednocześnie pracuje tylko jeden kompresor.
// stored: AutoNumber true, IsIECCheckEnabled false, IsRetainMemResEnabled false, MemoryReserve 500, SetENOAutomatically false, UDAEnableTagReadback false
   VAR_INPUT
      IsReadyP1 : Bool;   // Gotowość pompy
      IsReadyP2 : Bool;   // Gotowość pompy
      IsReadyP3 : Bool;   // Gotowość pompy
      IsReadyP4 : Bool;
      IsMode_Auto : Bool;   // Tryb pracy Aut
      InputWarning_H_PID : Bool;   // Oszczerzenie górny limit
      InputWarning_L_PID : Bool;   // Oczszczerzenie dolny limit
      IsReady_Inverter : Bool;   // Gotowość falownika
      PV_max : Real;   // Wartość górnego progu ostrzegawczego
      Act_B3ciśnienie : Real;   // Aktualna wartość bar
      Rst_Driver_Max_presure : Bool;   // Znacznika awaryjnego wyłączenia od max ciśnienia napędu pracującego w trybie awaryjnym
   END_VAR
   VAR_OUTPUT
      CMD_A_Network_P1 : Bool;   // Bit startu pompyw trybie awaryjnym na soft-startcie
      CMD_A_Network_P2 : Bool := false;   // Bit startu pompyw trybie awaryjnym na soft-startcie
      CMD_A_Network_P3 : Bool := false;   // Bit startu pompyw trybie awaryjnym na soft-startcie
      CMD_A_Network_P4 : Bool := false;   // Bit startu pompyw trybie awaryjnym na soft-startcie
   END_VAR
   VAR
      stc_PV : Real := 0.2;   // Ustalona wartość pomniejszenia PV
   END_VAR
   VAR_TEMP
      set_Motor : Bool;   // pomocniczy bit ustawiający pompę
      tmp_PVmax : Real;   // Tymczasowa ustalona wartość progu górnego bar
   END_VAR
BEGIN

REGION Network 2: Górny próg tymczasowy
   // Wyliczenie górnego progu tymczasowego na potrzeby sterowania wyłączaniem kompresora
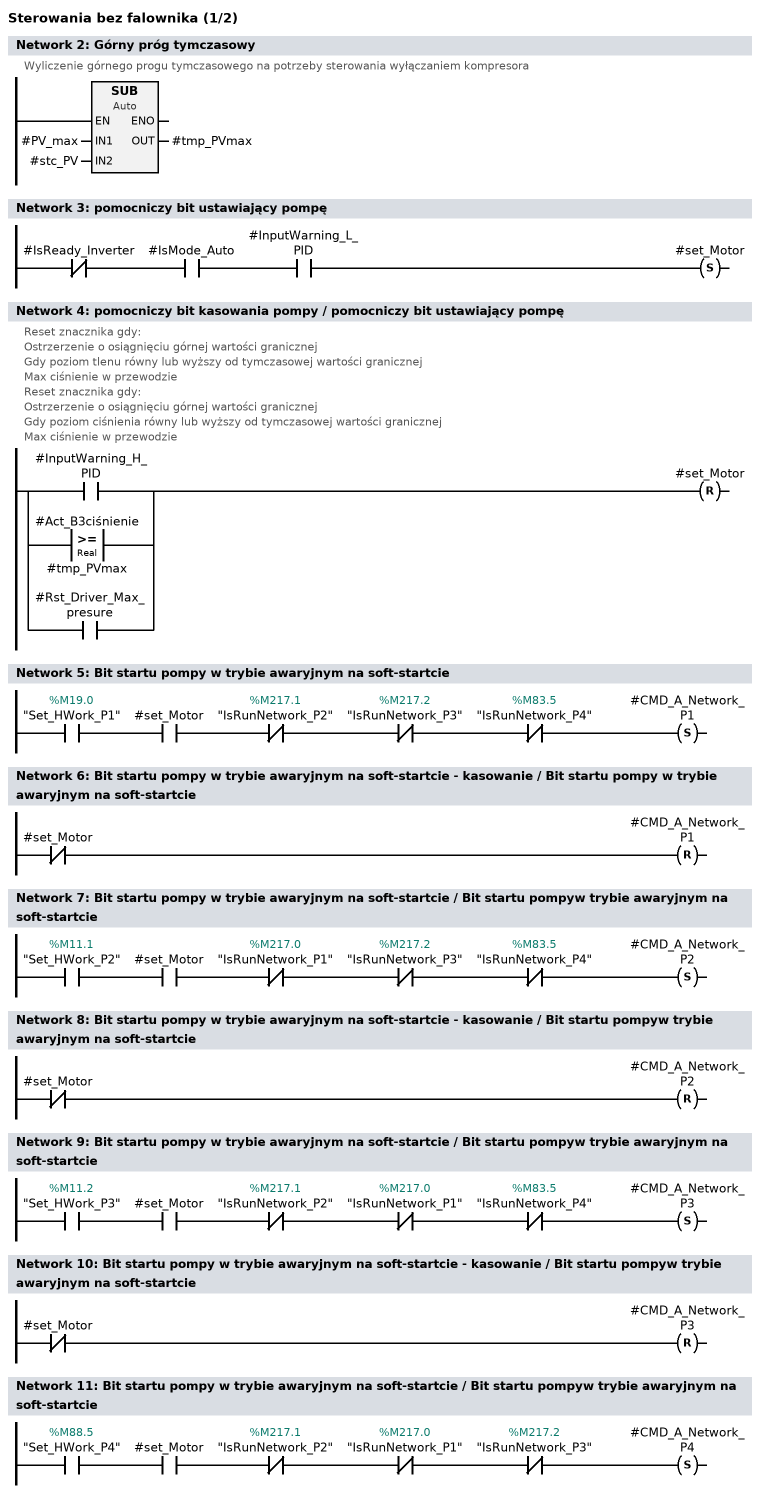
   RUNG wire#powerrail
      Sub(in1 := #PV_max, in2 := #stc_PV, out => #tmp_PVmax)
   END_RUNG
   // the same network as SCL:
   #tmp_PVmax := #PV_max - #stc_PV;
END_REGION

REGION Network 3: pomocniczy bit ustawiający pompę
   RUNG wire#powerrail
      I_Contact( #IsReady_Inverter )
      Contact( #IsMode_Auto )
      Contact( #InputWarning_L_PID )
      S_Coil( #set_Motor )
   END_RUNG
   // the same network as SCL:
   IF NOT #IsReady_Inverter AND #IsMode_Auto AND #InputWarning_L_PID THEN #set_Motor := TRUE; END_IF;
END_REGION

REGION Network 4: pomocniczy bit kasowania pompy / pomocniczy bit ustawiający pompę
   // Reset znacznika gdy:
   // Ostrzerzenie o osiągnięciu górnej wartości granicznej
   // Gdy poziom tlenu równy lub wyższy od tymczasowej wartości granicznej
   // Max ciśnienie w przewodzie
   // Reset znacznika gdy:
   // Ostrzerzenie o osiągnięciu górnej wartości granicznej
   // Gdy poziom ciśnienia równy lub wyższy od tymczasowej wartości granicznej
   // Max ciśnienie w przewodzie
   RUNG wire#powerrail
      Contact( #InputWarning_H_PID )
      wire#w1
      R_Coil( #set_Motor )
   END_RUNG
   RUNG wire#powerrail
      { S7_Templates := "SrcType := Real" } GE_Contact(in1 := #Act_B3ciśnienie, in2 := #tmp_PVmax)
   END_RUNG wire#w1
   RUNG wire#powerrail
      Contact( #Rst_Driver_Max_presure )
   END_RUNG wire#w1
   // the same network as SCL:
   IF #InputWarning_H_PID OR (#Act_B3ciśnienie >= #tmp_PVmax) OR #Rst_Driver_Max_presure THEN
       #set_Motor := FALSE;
   END_IF;
END_REGION

REGION Network 5: Bit startu pompy w trybie awaryjnym na soft-startcie
   RUNG wire#powerrail
      Contact( "Set_HWork_P1" )
      Contact( #set_Motor )
      I_Contact( "IsRunNetwork_P2" )
      I_Contact( "IsRunNetwork_P3" )
      I_Contact( "IsRunNetwork_P4" )
      S_Coil( #CMD_A_Network_P1 )
   END_RUNG
   // the same network as SCL:
   IF "Set_HWork_P1" AND #set_Motor AND NOT "IsRunNetwork_P2" AND NOT "IsRunNetwork_P3" AND NOT "IsRunNetwork_P4" THEN
       #CMD_A_Network_P1 := TRUE;
   END_IF;
END_REGION

REGION Network 6: Bit startu pompy w trybie awaryjnym na soft-startcie - kasowanie / Bit startu pompy w trybie awaryjnym na soft-startcie
   RUNG wire#powerrail
      I_Contact( #set_Motor )
      R_Coil( #CMD_A_Network_P1 )
   END_RUNG
   // the same network as SCL:
   IF NOT #set_Motor THEN #CMD_A_Network_P1 := FALSE; END_IF;
END_REGION

REGION Network 7: Bit startu pompy w trybie awaryjnym na soft-startcie / Bit startu pompyw trybie awaryjnym na soft-startcie
   RUNG wire#powerrail
      Contact( "Set_HWork_P2" )
      Contact( #set_Motor )
      I_Contact( "IsRunNetwork_P1" )
      I_Contact( "IsRunNetwork_P3" )
      I_Contact( "IsRunNetwork_P4" )
      S_Coil( #CMD_A_Network_P2 )
   END_RUNG
   // the same network as SCL:
   IF "Set_HWork_P2" AND #set_Motor AND NOT "IsRunNetwork_P1" AND NOT "IsRunNetwork_P3" AND NOT "IsRunNetwork_P4" THEN
       #CMD_A_Network_P2 := TRUE;
   END_IF;
END_REGION

REGION Network 8: Bit startu pompy w trybie awaryjnym na soft-startcie - kasowanie / Bit startu pompyw trybie awaryjnym na soft-startcie
   RUNG wire#powerrail
      I_Contact( #set_Motor )
      R_Coil( #CMD_A_Network_P2 )
   END_RUNG
   // the same network as SCL:
   IF NOT #set_Motor THEN #CMD_A_Network_P2 := FALSE; END_IF;
END_REGION

REGION Network 9: Bit startu pompy w trybie awaryjnym na soft-startcie / Bit startu pompyw trybie awaryjnym na soft-startcie
   RUNG wire#powerrail
      Contact( "Set_HWork_P3" )
      Contact( #set_Motor )
      I_Contact( "IsRunNetwork_P2" )
      I_Contact( "IsRunNetwork_P1" )
      I_Contact( "IsRunNetwork_P4" )
      S_Coil( #CMD_A_Network_P3 )
   END_RUNG
   // the same network as SCL:
   IF "Set_HWork_P3" AND #set_Motor AND NOT "IsRunNetwork_P2" AND NOT "IsRunNetwork_P1" AND NOT "IsRunNetwork_P4" THEN
       #CMD_A_Network_P3 := TRUE;
   END_IF;
END_REGION

REGION Network 10: Bit startu pompy w trybie awaryjnym na soft-startcie - kasowanie / Bit startu pompyw trybie awaryjnym na soft-startcie
   RUNG wire#powerrail
      I_Contact( #set_Motor )
      R_Coil( #CMD_A_Network_P3 )
   END_RUNG
   // the same network as SCL:
   IF NOT #set_Motor THEN #CMD_A_Network_P3 := FALSE; END_IF;
END_REGION

REGION Network 11: Bit startu pompy w trybie awaryjnym na soft-startcie / Bit startu pompyw trybie awaryjnym na soft-startcie
   RUNG wire#powerrail
      Contact( "Set_HWork_P4" )
      Contact( #set_Motor )
      I_Contact( "IsRunNetwork_P2" )
      I_Contact( "IsRunNetwork_P1" )
      I_Contact( "IsRunNetwork_P3" )
      S_Coil( #CMD_A_Network_P4 )
   END_RUNG
   // the same network as SCL:
   IF "Set_HWork_P4" AND #set_Motor AND NOT "IsRunNetwork_P2" AND NOT "IsRunNetwork_P1" AND NOT "IsRunNetwork_P3" THEN
       #CMD_A_Network_P4 := TRUE;
   END_IF;
END_REGION

